# B&R Automation Studio project MotionTestBenchMaster
Automation Studio 4.2.12.129 SP

## Logical view

Binary libraries used (declarations not repeated): ArEventLog, AsARCfg, AsArProf, AsArSdm, AsEthIP, AsIecCon, AsICMP, AsIODiag, AsMath, asstring, AsTCP, astime, AsUDP, brsystem, DataObj, FileIO, LoopConR 4.01.0, operator, powerlnk, runtime, standard, sys_lib, AsMem, AsBrStr, dvframe, MpRecipe 1.61.0, AsEPL, MpCom 1.61.0, AsXml, AsIOLink, AsIOAcc, Acp10man 3.17.2, Acp10par 3.17.2, NcGlobal 3.17.2, Acp10sim 3.17.2, Acp10_MC 3.17.2, MpAxis 1.61.0, MpAlarmX 1.61.0, MpWebXs 1.61.0

### Package Logical/00_AID - Aid memory: memorie ausiliarie al programma

### Program Logical/00_AID/AID (IEC) - AID Main Program - C#3 - 1.6ms

#### AID.st - Cyclic code
```iecst
PROGRAM _INIT
	AID.DataOut.ProjectType	:= CST_AID_ProjectMachine;
END_PROGRAM

PROGRAM _CYCLIC
	TimeAndBlink;

	Beacon_SidelStandard;

	PbLight;

	AID.DataOut.Reset		:= IO_PB_ResetOp.ON;//v4 200.2.0
	IO_SkdReset.DO_Output	:= AID.DataOut.Reset;

	IF EDGEPOS(IO_PB_ResetOp.ON) THEN
		AID.DataOut.OperatorPresence	:= TRUE;
	END_IF
END_PROGRAM
```

#### Variables.var - Local variables
```iecst
VAR
	TMR_TP_HornAlarmStop : TP_Reset;
	VAR_AlarmLightReset : BOOL;
	VAR_CriticalLight : BOOL;
	VAR_AlarmLight : BOOL;
	VAR_AlarmHorn : BOOL;
	FB_Blink_05Hz : FB_Blinker;
	FB_Blink_1Hz : FB_Blinker;
	FB_Blink_4Hz : FB_Blinker;
	FB_Blink_2Hz : FB_Blinker;
	VAR_RedLightFix : BOOL;
	VAR_RedLightFlash : BOOL;
	VAR_BlueLightFix : BOOL;
	VAR_BlueLightFlash : BOOL;
	TMR_TON_InterCpuCycleOk : TON;
END_VAR
```

### Global.typ - Global data types
```iecst
(*HMI/IO BOTTON TYPE*)

TYPE
	PB_Type : 	STRUCT  (*Push button (ON-OFF;) 0=OFF - 1=ON*)
		Enable : BOOL; (*State: Command Enabled*)
		LampON : BOOL; (*State: Lamp Command ON*)
		Blink : BOOL; (*State: Blink LampOn*)
		Visibility : BOOL; (*Configuration: Present*)
		ON : BOOL; (*Command: Push Button ON*)
	END_STRUCT;
	SS2P_Type : 	STRUCT  (*Selector 2 position (Auto-Man; ON-OFF;) 0=Auto/OFF - 1=Man/ON*)
		Enable : BOOL; (*State: Command Enabled*)
		LampON : BOOL; (*State: Lamp Command ON*)
		Blink : BOOL; (*State: Blink LampOn*)
		Visibility : BOOL; (*Configuration: Present*)
		ON : BOOL; (*Command: Selector Button ON*)
	END_STRUCT;
	SS3P_Type : 	STRUCT  (*Selector 3 position (Auto-0-Man)*)
		Enable : BOOL; (*State: Command Enabled*)
		LampON : BOOL; (*State: Lamp Command ON*)
		Blink : BOOL; (*State: Blink LampOn*)
		Visibility : BOOL; (*Configuration: Present*)
		Auto : BOOL := TRUE; (*Command: Automatic Mode*)
		Man : BOOL; (*Command: Manual Mode ON*)
	END_STRUCT;
	CmdBarPB_Type : 	STRUCT  (*Push button (ON-OFF;) 0=OFF - 1=ON*)
		Enable : BOOL; (*State: Command Enabled*)
		LampON : BOOL; (*State: Lamp Command ON*)
		Blink : BOOL; (*State: Blink LampOn*)
		Visibility : BOOL; (*Configuration: Present*)
		ON : BOOL; (*Command: Push Button ON*)
		Command : BOOL; (*Command: Push Button On from HMI OR Command from ITC*)
	END_STRUCT;
	SS2PCustom_Type : 	STRUCT  (*V4.A.A.1.6.13*)
		Enable : BOOL; (*State: Command Enabled*)
		LampON : BOOL; (*State: Lamp Command ON*)
		Blink : BOOL; (*State: Blink LampOn*)
		Visibility : BOOL; (*Configuration: Present*)
		ON : BOOL; (*Command: Selector Button ON*)
		Description : STRING[25];
	END_STRUCT;
END_TYPE

(*OUTPUT TYPE*)

TYPE
	IO_Beacon_Type : 	STRUCT
		DO_LightGreen : BOOL;
		DO_LightYellow : BOOL;
		DO_LightBlue : BOOL;
		DO_LightWhite : BOOL;
		DO_LightRed : BOOL;
		DO_Horn : BOOL;
	END_STRUCT;
END_TYPE
```

### Alarm.var - Alarms structure declaration
```iecst
VAR
	ALR : ARRAY[1..8000] OF AlarmCmd_Type;
	ALR_OldStatus : ARRAY[1..8000] OF BOOL;
	ALR_CFG : ARRAY[1..8000] OF AlarmCFG_Type;
	VAR_ALR_FirstAlertAlarmActive : AlarmCFG_Type; (*V4.A.A.1.7.0*)
	VAR_ALR_FirstCriticalAlarmActive : AlarmCFG_Type; (*V4.A.A.1.7.0*)
	VAR_ALR_FirstAlarmActive : AlarmCFG_Type; (*V4.A.A.1.7.0*)
	VAR_ALR_FirstExternalAlarmActive : AlarmCFG_Type; (*V4.A.A.1.7.0*)
	VAR_ALR_FirstExtCritAlarmActive : AlarmCFG_Type; (*V4.A.A.1.7.0*)
	VAR_ALR_FirstExtAlertAlarmActive : AlarmCFG_Type; (*V4.A.A.1.7.0*)
	VAR_ALR_FirstCsAlarmActive : AlarmCFG_Type; (*V4.A.A.1.7.0*)
	VAR_ALR_FirstCsExtAlarmActive : AlarmCFG_Type; (*V4.A.A.1.7.5a*)
	VAR_ALR_CriticalAcknoledgeReq : BOOL;
	VAR_ALR_AlarmAcknoledgeReq : BOOL;
	VAR_AlarmActionOper : ActionSum_Type; (*V4.A.A.1.6.13*)
	VAR_FMC_AlarmActionOper : ActionSum_Type;
	VAR_SKD_AlarmActionOper : ActionSum_Type;
END_VAR
```

### Package Logical/00_AID/IO - Input/Output declaration

### IO_AID.var
```iecst
VAR
	IO_SkdReset : IO_Digital_OUT_Type;
	IO_InterCpu_NettimeSoC : DINT;
	IO_InterCpu_CicleOk : BOOL;
END_VAR
```

### IO_CAP.var
```iecst
(*MOTORS*)
VAR
	IO_206MMR : IO_Motor_Type; (*Head rotation motor*)
	IO_206MMRBrake : IO_Motor_Type; (*Head rotation motor brake*)
	IO_207MMR : IO_Motor_Type; (*Hopper motor chute 1*)
	IO_211MMR : IO_Motor_Type; (*Buffer rotation motor2 v1.7.4*)
	IO_212MMR : IO_Motor_Type; (*Buffer rotation motor*)
	IO_213MMR : IO_Motor_Type; (*Head rotation motor fun*)
	IO_214MMR : IO_Motor_Type; (*Hopper motor chute 2*)
	IO_215MMR : IO_Motor_Type; (*Hopper motor chute 3*)
	IO_229MMR : IO_Motor_Type; (*Adjustment panel motor //V4.A.A.1.6.11*)
	IO_229MMR_Start : IO_SiriusStarter_Type; (*Adjustment panel motor //V4.A.A.1.6.11*)
	IO_230MMR : IO_Motor_Type; (*Dust removal motor on caps channel*)
	IO_231MMR : IO_Motor_Type; (*Dust removal motor on buffer //V4.A.A.1.6.11*)
	IO_202GPE : IO_GreasingPump_Type; (*Capper Greasing Motor*)
	IO_203GPE : IO_GreasingPump_Type; (*Capper Greasing Motor2 //V4.A.A.1.6.11*)
END_VAR
(*IONIZER*)
VAR
	IO_201DRC : IO_Motor_Type; (*Hopper motor chute 2*)
	IO_201DRC_SwitchFeedback : IO_Digital_IN_Type;
END_VAR
(*UV LAMP*)
VAR
	IO_201LLC : IO_Motor_Type; (*UV lamp Chute 1*)
	IO_202LLC : IO_Motor_Type; (*UV lamp Chute 2*)
	IO_203LLC : IO_Motor_Type; (*UV lamp Chute 3*)
END_VAR
(*DRIVERS*)
VAR
	IO_VFD_206MMR : IO_PLK_Danfoss_Drive_Type; (*Head rotation motor*)
	IO_VFD_207MMR : IO_PLK_Danfoss_Drive_Type; (*Hopper motor chute 1*)
	IO_VFD_230MMR : IO_PLK_Danfoss_Drive_Type; (*Dust remover motor*)
	IO_VFD_231MMR : IO_PLK_Danfoss_Drive_Type; (*Dust remover motor2 v1.7.4*)
	IO_VFD_211MMR : IO_PLK_Danfoss_Drive_Type; (*Buffer rotation motor2 v1.7.4*)
	IO_VFD_213MMR : IO_PLK_Danfoss_Drive_Type; (*Head rotation motor fun*)
	IO_VFD_212MMR : IO_PLK_Danfoss_Drive_Type; (*Buffer rotation motor*)
	IO_VFD_214MMR : IO_PLK_Danfoss_Drive_Type; (*Hopper motor chute 2*)
	IO_VFD_215MMR : IO_PLK_Danfoss_Drive_Type; (*Hopper motor chute 3*)
END_VAR
(*VALVES*)
VAR
	IO_201CPC : IO_Valve_Type; (*EV chute 1 caps release*)
	IO_202CPC : IO_Valve_Type; (*EV chute 2 caps release*)
	IO_205CPC : IO_Valve_Type; (*EV caps block chute 1*)
	IO_206CPC : IO_Valve_Type; (*EV caps block chute 2*)
	IO_207CPC : IO_Valve_Type; (*EV cap discharge door*)
	IO_212CPC : IO_Valve_Type; (*EV open buffer discharge door*)
	IO_213CPC : IO_Valve_Type; (*EV buffer lifting*)
	IO_214CPC : IO_Valve_Type; (*EV buffer lock*)
	IO_215CPC : IO_Valve_Type; (*EV lock size change guide*)
	IO_216CPC : IO_Valve_Type; (*EV 3 size change guide*)
	IO_217CPC : IO_Valve_Type; (*EV 4 size change guide*)
	IO_218CPC : IO_Valve_Type; (*EV sport size change guide*)
	IO_219CPC : IO_Valve_Type; (*EV open channel discharge door*)
	IO_220CPC : IO_Valve_Type; (*FREE v1.7.6*)
	IO_221CPC : IO_Valve_Type; (*EV chute 3 caps release*)
	IO_222CPC : IO_Valve_Type; (*EV caps block chute 3*)
	IO_223CPC : IO_Valve_Type; (*EV buffer vibrator*)
	IO_224CPC : IO_Valve_Type; (*EV cam position*)
	IO_225CPC : IO_Valve_Type; (*EV cam locking*)
	IO_226CPC : IO_Valve_Type; (*EV opening door UV Lamp A  V. 1.1*)
	IO_227CPC : IO_Valve_Type; (*EV  Block Caps Outlet Chute 1*)
	IO_228CPC : IO_Valve_Type; (*EV transfer Starwheel air soleniod valve DA VERIFICARE*)
	IO_229CPC : IO_Valve_Type; (*EV transfer Starwheel air soleniod valve DA VERIFICARE*)
	IO_232CPC : IO_Valve_Type; (*EV opening door UV Lamp B  V. 1.1*)
	IO_233CPC : IO_Valve_Type; (*EV opening door UV Lamp B  //V4.A.A.1.6.12*)
	IO_234CPC : IO_Valve_Type; (*EV Caps Ejection Cap Feeder   V4.A.A.1.7.1*)
	IO_235CPC : IO_Valve_Type; (*EV Caps Block Outlet Chuter2 //v1.7.4*)
	IO_236CPC : IO_Valve_Type; (*v1.7.4*)
	IO_237CPC : IO_Valve_Type; (*v1.7.4*)
	IO_238CPC : IO_Valve_Type; (*v1.7.4*)
	IO_201EVC : IO_Valve_Type; (*Air blowing for cap release 1 V 1.6*)
	IO_203EVC : IO_Valve_Type; (*Air blowing for cap release 2 V 1.6*)
	IO_207EVC : IO_Valve_Type; (*Air blowing for cap release 3 V 1.6*)
	IO_209EVC : IO_Valve_Type; (*FREE V1.6*)
	IO_210EVC : IO_Valve_Type; (*Air blowing for buffer emptying*)
	IO_211EVC : IO_Valve_Type; (*Buffer air blowing for caps release*)
	IO_212EVC : IO_Valve_Type; (*Air blowing for chute emptying*)
	IO_213EVC : IO_Valve_Type; (*Air blowing caps ionizer chute 1*)
	IO_214EVC : IO_Valve_Type; (*Air blowing caps ionizer chute 2*)
	IO_215EVC : IO_Valve_Type; (*Air blowing caps ionizer chute 3*)
	IO_216EVC : IO_Valve_Type; (*Air blowing for chute emptying by PeP*)
	IO_227EVC : IO_Valve_Type; (*v1.7.4*)
	IO_228EVC : IO_Valve_Type; (*v1.7.4*)
	IO_229EVC : IO_Valve_Type; (*v1.7.4*)
	IO_203EVF : IO_Valve_Type; (*Air blowing caps (Drying)*) (*IO_AVC : ARRAY[MIN_CFG_AVC..MAX_CFG_AVC] OF IO_Valve_Type; Caps Treatment Valves v4.A.A.1.7.0*)
END_VAR
(*SENSOR*)
VAR
	IO_201DSC : IO_Digital_IN_Type; (*Caps/crowns release check*)
	IO_202DSC : IO_Digital_IN_Type; (*Low level caps/crowns presence chute 1*)
	IO_204DSC : IO_Digital_IN_Type; (*Head 1 sensor*)
	IO_205DSC : IO_Digital_IN_Type; (*Lack of caps (Quibuf infeed)*)
	IO_210DSC : IO_Digital_IN_Type; (*Cap Overturned hight Cap Feeder  V4.A.A.1.7.1*)
	IO_211DSC : IO_Digital_IN_Type; (*Cap Overturned low Cap Feeder  V4.A.A.1.7.1*)
	IO_216DSC : IO_Digital_IN_Type; (*Low level caps/crowns presence chute 2*)
	IO_217DSC : IO_Digital_IN_Type; (*Low level caps/crowns presence chute 3*)
	IO_218DSC : IO_Digital_IN_Type; (*Upside down caps check chute 1 high*)
	IO_219DSC : IO_Digital_IN_Type; (*Upside down caps check chute 1 low*)
	IO_220DSC : IO_Digital_IN_Type; (*Upside down caps check chute 2 high*)
	IO_221DSC : IO_Digital_IN_Type; (*Upside down caps check chute 2 low*)
	IO_222DSC : IO_Digital_IN_Type; (*Upside down caps check chute 3 high*)
	IO_223DSC : IO_Digital_IN_Type; (*Upside down caps check chute 3 low*)
	IO_224DSC : IO_Digital_IN_Type; (*Ionizer pressure switch chute 1*)
	IO_225DSC : IO_Digital_IN_Type; (*Ionizer pressure switch chute 2*)
	IO_226DSC : IO_Digital_IN_Type; (*Ionizer pressure switch chute 3*)
	IO_227DSC : IO_Digital_IN_Type; (*Lubrication door sensor*)
	IO_228DSC : IO_Digital_IN_Type; (*Fixed part lubrication check*)
	IO_229DSC : IO_Digital_IN_Type; (*Rotating part lubrication check*)
	IO_230DSC : IO_Digital_IN_Type; (*Lubrication pipe inserted sensor*)
	IO_231DSC : IO_Digital_IN_Type; (*Turret cam position analog sensor*)
	IO_232DSC : IO_Digital_IN_Type; (*Caps buffer full*)
	IO_233DSC : IO_Digital_IN_Type; (*Caps channel discharge gate sensor*)
	IO_234DSC : IO_Digital_IN_Type; (*Lubrication phase sensor*)
	IO_235DSC : IO_Digital_IN_Type; (*Buffer in high position*)
	IO_236DSC : IO_Digital_IN_Type; (*Buffer in low position*)
	IO_237DSC : IO_Digital_IN_Type; (*Buffer lock inserted*)
	IO_238DSC : IO_Digital_IN_Type; (*Caps buffer max level chute 1*)
	IO_239DSC : IO_Digital_IN_Type; (*Caps buffer max level chute 2*)
	IO_240DSC : IO_Digital_IN_Type; (*Caps buffer max level chute 3*)
	IO_241DSC : IO_Digital_IN_Type; (*Hopper level chute 1*)
	IO_242DSC : IO_Digital_IN_Type; (*Hopper level chute 2*)
	IO_243DSC : IO_Digital_IN_Type; (*Hopper level chute 3*)
	IO_244DSC : IO_Digital_IN_Type; (*Max level caps/crowns chute 1*)
	IO_245DSC : IO_Digital_IN_Type; (*Max level caps/crowns chute 2*)
	IO_246DSC : IO_Digital_IN_Type; (*Max level caps/crowns chute 3*)
	IO_247DSC : IO_Digital_IN_Type; (*Medium level caps/crowns chute 1*)
	IO_248DSC : IO_Digital_IN_Type; (*Medium level caps/crowns chute 2*)
	IO_249DSC : IO_Digital_IN_Type; (*Medium level caps/crowns chute 3*)
	IO_250DSC : IO_Digital_IN_Type; (*Side door hopper sport*)
	IO_251DSC : IO_Digital_IN_Type; (*Top door hopper sport*)
	IO_252DSC : IO_Digital_IN_Type; (*Uv lamp door*)
	IO_253DSC : IO_Digital_IN_Type; (*Sensore carter posteriore*)
	IO_254DSC : IO_Digital_IN_Type; (*Sensore di fase per lubrificazione*)
	IO_255DSC : IO_Digital_IN_Type; (*Sensore di lubrificazione della parte fissa*)
	IO_256DSC : IO_Digital_IN_Type; (*Sensore di lubrificazione della parte rotante*)
	IO_257DSC : IO_Digital_IN_Type; (*Sensore di inserimento del raccordo di lubrificazione della parte rotante *)
	IO_258DSC : IO_Digital_IN_Type; (*Sensore carter superiore  //V4.A.A.1.6.11*)
	IO_259DSC : IO_Digital_IN_Type; (*Sensore di lubrificazione rotazione teste //V4.A.A.1.6.11*)
	IO_260DSC : IO_Digital_IN_Type; (*Sensore di inserimento del raccordo di lubrificazione della parte rotante riduttore rotazione teste //V4.A.A.1.6.11*)
	IO_261DSC : IO_Digital_IN_Type; (*Sensore limite minimo posizione pannello //V4.A.A.1.6.11*)
	IO_262DSC : IO_Digital_IN_Type; (*Sensore zero encoder //V4.A.A.1.6.11*)
	IO_263DSC : IO_Digital_IN_Type; (*Sensore limite massimo posizione pannello //V4.A.A.1.6.11*)
	IO_264DSC : IO_Digital_IN_Type; (*Caps/Crown release check on bottle   //V4.A.A.1.6.12h*)
	IO_266DSC : IO_Digital_IN_Type; (*Flow Cap Control //v1.7.4*)
	IO_267DSC : IO_Digital_IN_Type; (*v1.7.5*)
	IO_268DSC : IO_Digital_IN_Type; (*v1.7.5*)
	IO_270DSC : IO_Digital_IN_Type; (*Caps Belt Sensor  //v1.7.4*)
	IO_ST3B : IO_Analog_IN_Type; (*Sensore temperatura motore//V4.A.A.1.6.12*)
	IO_ST3A : IO_Analog_IN_Type; (*Sensore temperatura motore//V4.A.A.1.6.12*)
END_VAR
(*COUNTERS*)
VAR
	IO_201DGC : IO_IncrementalEncoder; (*Incremental Encoder adjustment panel //V4.A.A.1.6.11*)
END_VAR
(*PB*)
VAR
	IO_PB_BufferUp : PB_Type;
	IO_PB_BufferDown : PB_Type;
END_VAR
(*MOTORS EQUATORQUE & HRM*)
VAR
	IO_BrushHead : IO_Motor_Type; (*Outfeed Conveyor Motor V4.A.A.1.6.12*)
END_VAR
(*DIGITAL OUTPUT*)
VAR
	IO_CAP_24Vdc_OK : IO_Digital_OUT_Type; (*v1.5*)
	IO_BottlePresence : IO_Digital_OUT_Type; (*v1.5*)
	IO_CapsRequest : IO_Digital_OUT_Type; (*v1.7.4 Richiesta capsule all'elevatore*)
END_VAR
```

### IO_CRW.var
```iecst
(*VALVES*)
VAR
	IO_230CPC : IO_Valve_Type; (*EV chute 1 crowns release*)
	IO_231CPC : IO_Valve_Type; (*EV chute 2 crowns release*)
	IO_231EVC : IO_Valve_Type;
	IO_205EVC : IO_Valve_Type; (*EXTRACTOR BLOWER CLEANING*)
	IO_274DSC : IO_Digital_IN_Type; (*Master nuovo*)
END_VAR
```

### IO_CSR.var
```iecst
(*Master nuovo*)
VAR
	IO_204CPC : IO_Valve_Type; (*EV crowner lift block*)
	IO_LTK : ARRAY[MIN_CFG_LTx..MAX_CFG_LTx] OF IO_Analog_IN_Type;
	IO_3281M1 : IO_Motor_FwBw_Type;
	IO_3281M1_Cmd : IO_Digital_OUT_Type;
	IO_2806M1 : IO_Motor_FwBw_Type;
	IO_2806M1_Cmd : IO_Digital_OUT_Type;
	IO_2808M1 : IO_Motor_FwBw_Type;
	IO_2806M1_Brake : IO_Motor_Type;
	IO_2809M2_Brake : IO_Motor_Type;
	IO_2809M2 : IO_Motor_FwBw_Type;
	IO_RnsLiftFC280 : IO_MotorFC280_Type; (*Rinser Lift*)
	IO_VFD_RnsLiftFC280 : IO_PLK_DanfossFC280_Drive_Type; (*Rinser Lift VFD*)
	IO_TnkLiftFC280 : IO_MotorFC280_Type;
	IO_VFD_TnkLiftFC280 : IO_PLK_DanfossFC280_Drive_Type; (*Outfeed Conveyor VFD*)
	IO_2768U0 : IO_Motor_FwBw_Type;
	IO_2768U0_Store : IO_Digital_OUT_Type;
	IO_202CPB : IO_Valve_Type; (*Containers sectors block (X: Block / Y: Unblock)*)
	IO_212DSB : IO_Digital_IN_Type; (*Third element perso part sensor*)
	IO_213DSB : IO_Digital_IN_Type; (*Third element perso part sensor - Ferrum Guide Presence in Carousel Outlet*)
	IO_CSR_SCU : IO_CSR_SCU_Type;
	IO_CSR_FlrShaftSensorCtrl1 : IO_Digital_IN_Type;
	IO_CSR_FlrShaftSensorCtrl2 : IO_Digital_IN_Type;
	IO_CSR_RnsShaftSensorCtrl1 : IO_Digital_IN_Type;
	IO_CSR_RnsShaftSensorCtrl2 : IO_Digital_IN_Type;
	IO_YV26 : IO_Valve_Type;
	IO_YV39 : IO_Valve_Type;
	IO_SQ26 : IO_Digital_IN_Type;
	IO_SQ45A2 : IO_Digital_IN_Type;
	IO_SQ45A1 : IO_Digital_IN_Type;
	IO_SQ70 : IO_Digital_IN_Type;
	IO_SQ5 : IO_Digital_IN_Type;
	IO_SQ40 : IO_Digital_IN_Type;
	IO_SQ6 : IO_Digital_IN_Type;
	IO_3565S5 : IO_Digital_IN_Type;
	IO_3565S7 : IO_Digital_IN_Type;
	IO_CapChannelPresent : IO_Digital_IN_Type;
END_VAR
(*SIKO*)
VAR
	IO_SIKO_AX2_SafetyEnable : IO_Digital_IN_Type := (DI_Input:=TRUE);
	IO_SIKO_AX1_SafetyEnable : IO_Digital_IN_Type := (DI_Input:=TRUE);
	IO_SIKO_AX1_Overload : IO_Digital_IN_Type := (DI_Input:=TRUE);
	IO_SIKO_AX2_Overload : IO_Digital_IN_Type := (DI_Input:=TRUE);
	IO_SIKO_AX1_ModuleOK : IO_Digital_IN_Type; (*Module Ok: Put this IO in The IoMap*)
	IO_SIKO_AX2_ModuleOK : IO_Digital_IN_Type; (*Module Ok: Put this IO in The IoMap*)
	IO_SIKO_AX1 : SIKO_COM_Type;
	IO_SIKO_AX2 : SIKO_COM_Type;
	IO_238DSE : IO_Digital_IN_Type; (*Outlet Conveyor Height Sensor*)
	IO_243DSE : IO_Digital_IN_Type; (*Outlet Conveyor Body Guide Presence*)
END_VAR
```

### IO_DMC.var
```iecst
VAR
	IO_210EVF : IO_Valve_Type; (*master nuovo*)
	IO_211EVF : IO_Valve_Type; (*master nuovo*)
	IO_RollSafety1 : IO_Dmc_Type;
	IO_RollSafety2 : IO_Dmc_Type;
	IO_DmcDevice : IO_Dmc_Type;
	IO_205DSF : IO_Digital_IN_Type; (*Dummy container inserted*)
END_VAR
```

### IO_FMC.var
```iecst
VAR
	IO_PB_FmcStartFilling : PB_Type; (*Manual filling start from Hw button*)
	IO_PB_FmcStopFilling : PB_Type; (*Manual filling stop from Hw button*)
	IO_PB_FmcStep : PB_Type; (*Single step from Hw button*)
END_VAR
```

### IO_GNS.var
```iecst
(*VALVES*)
VAR
	IO_201EVR : IO_Valve_Type; (*Ev MB05 Cooling*)
	IO_204EVF : IO_Valve_Type; (*Ev Pilot valve air (X: Discharge / Y: Charge)*)
	IO_205EVF : IO_Valve_Type;
END_VAR
(*SENSORS*)
VAR
	IO_204PSF : IO_Digital_IN_Type; (*Carousel air pressure switch*)
	IO_201PTF : IO_Analog_IN_Type; (*Carousel air pressure sensor*)
	IO_205PTF : IO_Analog_IN_Type; (*Carousel air pressure sensor*)
	IO_206PTF : IO_Analog_IN_Type; (*Carousel air pressure sensor*)
	IO_204PTF : IO_Analog_IN_Type; (*Carousel air pressure sensor*)
	IO_235DSE : IO_Digital_IN_Type; (*Cop mode Conveyor Outlet*)
	IO_239DSE : IO_Digital_IN_Type; (*Production mode Transfer Inlet*)
	IO_240DSE : IO_Digital_IN_Type; (*Cop mode Transfer Inlet*)
	IO_242DSE : IO_Digital_IN_Type; (*Production mode Conveyor Outlet*)
	IO_ContainerBurst1 : IO_Digital_IN_Type; (*ContainerBurst#1*)
	IO_ContainerBurst2 : IO_Digital_IN_Type; (*ContainerBurst#2 *)
	IO_201QTB : IO_Analog_IN_Type; (*Basement Air Control - CO2 Sensor //v1.7.4*)
	IO_201QTB_Warning : IO_Digital_IN_Type; (*Basement Air Control - CO2 Sensor Warning //v1.7.4*)
	IO_201QTB_Alarm : IO_Digital_IN_Type; (*Basement Air Control - CO2 Sensor Alarm//v1.7.4*)
	IO_201QTE : IO_Analog_IN_Type; (*Filler Air Control - CO2 Sensor //v1.7.4*)
	IO_201QTE_Warning : IO_Digital_IN_Type; (*FIller Air Control - CO2 Sensor Warning //v1.7.4*)
	IO_201QTE_Alarm : IO_Digital_IN_Type; (*Filler Air Control - CO2 Sensor Alarm//v1.7.4*)
	IO_202QTB : IO_Analog_IN_Type; (*Basement Air Control - Ozozne Sensor //v1.7.4*)
	IO_202QTB_Warning : IO_Digital_IN_Type; (*Basement Air Control - Ozozne Sensor Warning //v1.7.4*)
	IO_202QTB_Alarm : IO_Digital_IN_Type; (*Basement Air Control - Ozozne Sensor Alarm//v1.7.4*)
	IO_202QTE : IO_Analog_IN_Type; (*Filler Air Control - Ozozne Sensor //v1.7.4*)
	IO_202QTE_Warning : IO_Digital_IN_Type; (*Filler Air Control - Ozozne Sensor Warning //v1.7.4*)
	IO_202QTE_Alarm : IO_Digital_IN_Type; (*Filler Air Control - Ozozne Sensor Alarm//v1.7.4*)
END_VAR
(*INSTRUMENTS - DIGITAL*)
VAR
	IO_MB05_Cooling : IO_Cooling_Type; (*MB05 Cooling*)
	IO_MB05_Overload : IO_Digital_IN_Type := (DI_Input:=TRUE); (*MB05 Auxiliary circuit ON*)
	IO_MB15_Cooling : IO_Cooling_Type; (*MB15 Cooling v1.62*)
	IO_MB15_Overload : IO_Digital_IN_Type := (DI_Input:=TRUE); (*MB15 Auxiliary circuit ON*)
	IO_MB25_Overload : IO_Digital_IN_Type := (DI_Input:=TRUE); (*MB25 Auxiliary circuit ON*)
	IO_MC01_Cooling : IO_Cooling_Type; (*MC01 Cooling*)
	IO_MC01_Overload : IO_Digital_IN_Type := (DI_Input:=TRUE); (*MC01 Auxiliary circuit ON*)
	IO_MC02_Cooling : IO_Cooling_Type; (*MC02 Cooling*)
	IO_MC02_5VOverload : IO_Digital_IN_Type := (DI_Input:=TRUE); (*MC02 Auxiliary circuit ON*)
	IO_MC02_Overload : IO_Digital_IN_Type := (DI_Input:=TRUE); (*MC02 Auxiliary circuit ON*)
	IO_MC04_Cooling : IO_Cooling_Type; (*MC04 Cooling*)
	IO_MC04_Overload : IO_Digital_IN_Type := (DI_Input:=TRUE); (*MC04 Auxiliary circuit ON*)
	IO_MC04_CabinetDoorsUnlockFbk : IO_Digital_IN_Type; (*MC04 Cabinet Doors Unlock Feedback*)
	IO_MC04_CabinetDoorsUnlockReq : IO_Digital_IN_Type; (*MC04 Cabinet Doors Unlock Request*)
	IO_MC04_DoorCabinetOpened : IO_Digital_IN_Type := (DI_Input:=TRUE); (*MC04 Cabinet Door Opened*)
	IO_MC07_Cooling : IO_Cooling_Type; (*MC07 Cooling*)
	IO_MC07_Overload : IO_Digital_IN_Type := (DI_Input:=TRUE); (*MC07 Auxiliary circuit ON*)
	IO_MC07_DoorCabinetOpened : IO_Digital_IN_Type := (DI_Input:=TRUE); (*MC07 Cabinet Door Opened*)
	IO_MC19_Overload : IO_Digital_IN_Type := (DI_Input:=TRUE); (*MC19 Auxiliary circuit ON*)
	IO_MC19_DoorCabinetOpened : IO_Digital_IN_Type := (DI_Input:=TRUE); (*MC19 Cabinet Door Opened*)
	IO_MC29_Cooling : IO_Cooling_Type; (*MC29 Cooling  //v999hema*)
	IO_MC29_Overload : IO_Digital_IN_Type := (DI_Input:=TRUE); (*MC29 Auxiliary circuit ON //v999hema*)
	IO_MC29_DoorCabinetOpened : IO_Digital_IN_Type := (DI_Input:=TRUE); (*MC29 Cabinet Door Opened VRMA*)
	IO_CapFeederOverload : IO_Digital_IN_Type := (DI_Input:=TRUE); (*CapFeeder Overload ON*)
	IO_OptifeedOverload : IO_Digital_IN_Type := (DI_Input:=TRUE); (*Optifeed Overload ON //V4.A.A.1.6.11*)
	IO_UPS : IO_UPS_Type;
END_VAR
(*OUTPUT*)
VAR
	IO_FlrBeacon : IO_Beacon_Type;
END_VAR
```

### IO_ITC.var
```iecst
VAR
	IO_PB_LbStart : PB_Type; (*Labeller start Hw button*)
	IO_PB_LbStop : PB_Type; (*Labeller stop Hw button*)
END_VAR
(*HARDWARE\DP COMMUNICATION*)
VAR
	IO_ITC : IO_ITC_Type;
END_VAR
```

### IO_MAU.var
```iecst
(*MOTORS*)
VAR
	IO_201GPE : IO_GreasingPump_Type; (*MACHINE GREASING PUMP*)
END_VAR
(*OUTPUT*)
VAR
	IO_MachineLight : IO_Digital_OUT_Type;
END_VAR
(*PRESSURIZER*)
VAR
	IO_FanBase : IO_FanMain_Type;
	IO_FanFiller : IO_FanMain_Type;
	IO_FanRinser : IO_FanMain_Type;
	IO_FanTransfer : IO_FanMain_Type;
END_VAR
(*PLC*)
VAR
	IO_CPU : IO_CPU_Type;
END_VAR
(*LIFT CONTAINERS*)
VAR
	IO_203PSF : IO_Digital_IN_Type;
	IO_205RVF : IO_Analog_IN_OUT_Type;
	IO_203RVF : IO_Analog_IN_OUT_Type;
	IO_206DSF : IO_Digital_IN_Type; (*Filling valve 1 sensor*)
	IO_FSF : ARRAY[MIN_CFG_FSx..MAX_CFG_FSx] OF IO_Digital_IN_Type;
END_VAR
```

### IO_MNM.var
```iecst
VAR
	IO_PB_FlStart : PB_Type; (*Filler start Hw button*)
	IO_PB_FlStop : PB_Type := (ON:=TRUE); (*Filler stop Hw button*)
	IO_PB_ResetOp : PB_Type; (*Reset Hw button*)
	IO_PB_ResetFwIn : PB_Type; (*Reset Hw button*)
	IO_PB_ResetFwOut : PB_Type; (*Reset Hw button*)
	IO_PB_ResetBkIn : PB_Type; (*Reset Hw button*)
	IO_PB_ResetBkOut : PB_Type; (*Reset Hw button*)
	IO_KochModuleOk : IO_Digital_IN_Type;
END_VAR
(*MOTORS*)
VAR
	IO_InCvrFC280 : IO_MotorFC280_Type; (*Outfeed Conveyor Motor*) (*Master nuovo*)
	IO_OutCvrFC280 : IO_MotorFC280_Type; (*Outfeed Conveyor Motor*) (*Master nuovo*)
	IO_InCvr : IO_Motor_Type; (*Outfeed Conveyor Motor*) (*Master nuovo*)
	IO_OutCvr : IO_Motor_Type; (*Outfeed Conveyor Motor*)
END_VAR
(*DRIVERS*)
VAR
	IO_VFD_InCvrFC280 : IO_PLK_DanfossFC280_Drive_Type; (*Outfeed Conveyor VFD*) (*Master nuovo*)
	IO_VFD_OutCvrFC280 : IO_PLK_DanfossFC280_Drive_Type; (*Outfeed Conveyor VFD*) (*Master nuovo*)
	IO_VFD_InCvr : IO_PLK_Danfoss_Drive_Type; (*Outfeed Conveyor VFD*) (*Master nuovo*)
	IO_VFD_OutCvr : IO_PLK_Danfoss_Drive_Type; (*Outfeed Conveyor VFD*)
END_VAR
(*DIGITAL INSTUMENTS*)
VAR
	IO_241DSE : IO_Digital_IN_Type; (*Caps Discharge*)
	IO_230DSE : IO_Digital_IN_Type; (*Spot safety*)
	IO_236DSE : IO_Digital_IN_Type; (*Outlet obstructed*)
	IO_217DSR : IO_Digital_IN_Type; (*Machine upper part access tool position control V4.A.A.1.6.13*)
	IO_296CPB_I : IO_Digital_IN_Type; (*V4.A.A.1.7.0 RInser Bypass Control*)
	IO_297CPB_I : IO_Digital_IN_Type; (*V4.A.A.1.7.0 Rinser Bypass Control*)
	IO_224DSB : IO_Digital_IN_Type; (*Doser Bypass Control RMH017*)
	IO_225DSB : IO_Digital_IN_Type; (*Doser Bypass Control *)
	IO_226DSB : IO_Digital_IN_Type; (*Doser Bypass Control *)
	IO_227DSB : IO_Digital_IN_Type; (*Doser Bypass Control *)
END_VAR
(*MOTION Feedback*)
VAR
	IO_MNM_MotionFan : IO_MotionFanMachine_Type;
	IO_MNM_PowerSupply1Overload : IO_Digital_IN_Type := (DI_Input:=TRUE);
	IO_MNM_PowerSupply2Overload : IO_Digital_IN_Type := (DI_Input:=TRUE);
END_VAR
(*INLET CANS SENSOR*)
VAR
	IO_InletSafetyLow1 : IO_Digital_IN_Type;
	IO_InletSafetyHigh1 : IO_Digital_IN_Type;
	IO_InletSafetyLow2 : IO_Digital_IN_Type;
	IO_InletSafetyHigh2 : IO_Digital_IN_Type;
END_VAR
(*INLET CONTAINER RESET*)
(*Master nuovo*)
VAR
	IO_PB_ResetInlet1 : PB_Type; (*Master nuovo*)
	IO_PB_ResetInlet2 : PB_Type; (*Master nuovo*)
END_VAR
(* *)
VAR
	IO_LimitTorqueBlowerTransfer : IO_Digital_IN_Type := (DI_Input:=TRUE);
END_VAR
```

### IO_MC.var
```iecst
VAR
	IO_MCRaw : IO_MCRaw_Type;
	ITC_Motion_ExtEncModuleOk : BOOL;
	ITC_Motion_ExtEnc : DINT;
END_VAR
```

### IO_OPS.var
```iecst
VAR
	PO : PO_Safety_Type;
	PI : PI_Safety_Type;
	IO_OPS_Door : ARRAY[MIN_CFG_SafetyZone..MAX_CFG_SafetyZone,MIN_CFG_SafetyDoor..MAX_CFG_SafetyDoor] OF IO_OPS_Door_Type; (*1: Forward
2: Backward 1
3: Backward 2
4: Inlet Transfer Forward
5: Inlet Transfer Backward
6: Outlet Transfer Forward
7: Outlet Transfer Backward
8: Maintenance 1
9: Maintenance 2
10: Inlet Transfer Gate
11: Outlet Transfer Gate
12: Capper*)
	IO_OPS_Zone : ARRAY[MIN_CFG_SafetyZone..MAX_CFG_SafetyZone] OF IO_OPS_Zone_Type; (*1: Forward
2: Backward 1
3: Backward 2
4: Inlet Transfer Forward
5: Inlet Transfer Backward
6: Outlet Transfer Forward
7: Outlet Transfer Backward
8: Maintenance 1
9: Maintenance 2
10: Inlet Transfer Gate
11: Outlet Transfer Gate
12: Capper*)
	IO_OPS_JOG : ARRAY[MIN_CFG_SafetyJog..MAX_CFG_SafetyJog] OF IO_OPS_JOG_Type;
	IO_207EVF : IO_Valve_Type; (*Soffio Paratia automatica COP V4.A.A.1.6.12*)
	IO_208CPF : IO_Valve_Type; (*Paratia automatica COP V4.A.A.1.6.12*)
	IO_208DSFX : IO_Digital_IN_Type; (*Paratia automatica COP Aperta V4.A.A.1.6.12*)
	IO_208DSFY : IO_Digital_IN_Type; (*Paratia automatica COP Chiusa V4.A.A.1.6.12*)
	IO_209DSFX : IO_Digital_IN_Type; (*Paratia automatica COP Aperta V4.A.A.1.6.12*)
	IO_209DSFY : IO_Digital_IN_Type; (*Paratia automatica COP Chiusa V4.A.A.1.6.12*)
	IO_209EVF : IO_Valve_Type;
	IO_SS3P_Modality : IO_SS3PModality_Type;
	SI_SafeLogicModuleOk : BOOL;
	IO_Euchner_Key : IO_Digital_IN_Type; (*V1.3*)
	IO_Euchner_Strobe : IO_Digital_IN_Type; (*V1.3*)
	IO_Euchner_CodeA : IO_Digital_IN_Type; (*V1.3*)
	IO_Euchner_CodeB : IO_Digital_IN_Type; (*V1.3*)
	IO_Euchner_CodeC : IO_Digital_IN_Type; (*V1.3*)
	IO_Euchner_CodeD : IO_Digital_IN_Type; (*V1.3*)
	IO_PB_FlrSlowRun1 : PB_Type; (*V1.3*)
	IO_PB_FlrSlowRun2 : PB_Type; (*V1.3*)
	IO_PB_FlrSlowRun3 : PB_Type; (*V1.3*)
END_VAR
```

### IO_SFT.var
```iecst
(*SENSORS*)
(*ANOLOG SENSORS*)
VAR
	IO_203DSF : IO_Digital_IN_Type; (*Container presence outlet filler*)
	IO_202DSF : IO_Digital_IN_Type; (*Filler inlet container presence*)
	IO_208FSE : IO_Digital_IN_Type; (*Washing Ramp3 Flow-switch*)
	IO_207FSE : IO_Digital_IN_Type; (*Washing Ramp2 Flow-switch*)
	IO_ProductionSensorCheck1 : IO_Digital_IN_Type; (*Production Sensor Check For DMC Automatic*) (*Master nuovo*)
	IO_ProductionSensorCheck2 : IO_Digital_IN_Type; (*Production Sensor Check For DMC Automatic*) (*Master nuovo*)
	IO_ProductionSensorCheck3 : IO_Digital_IN_Type; (*Production Sensor Check For DMC Automatic*) (*Master nuovo*)
END_VAR
(*FLOW-SWITCHES*)
VAR
	IO_206FSE : IO_Digital_IN_Type; (*Washing Ramp1 Flow-switch*)
	IO_202EVR : IO_Valve_Type; (*Ev guide heater (VBS)*)
	IO_208CPB : IO_Valve_Type; (*Nob Nos 2° Treatment*)
	IO_207CPB : IO_Valve_Type; (*Nob Nos 1° Treatment*)
	IO_207CPF : IO_Valve_Type; (*Roller Security Cam*)
END_VAR
(*VALVES*)
VAR
	IO_201CPB : IO_Valve_Type; (*Inlet Bottle Block Bottle Stop*)
	IO_BurstCheck : ARRAY[0..2] OF IO_Digital_IN_Type; (*Container Burst Check 1*) (*Master nuovo*)
	IO_205DSB : IO_Digital_IN_Type; (*Doser outlet container presence*)
	IO_208DSF : IO_Digital_IN_Type; (*Rinser outlet container presence*)
	IO_DummyClock : IO_Digital_IN_Type; (*Rinser inlet container presence*)
	IO_207DSF : IO_Digital_IN_Type; (*Rinser inlet container presence*)
	IO_204DSF : IO_Digital_IN_Type; (*Container presence for filling valve opening*)
	IO_201DSF : IO_Digital_IN_Type; (*Filling valve 1 sensor*)
	IO_214DSF : IO_Digital_IN_Type; (*Head 1 Pulp Doser sensor //v999hema*)
	IO_204DSB : IO_Digital_IN_Type; (*Doser inlet container presence //v999hema*)
	IO_210CPF : IO_Valve_Type; (*Pulp Doser Pulp Valve Opening //v999hema*)
END_VAR
```

### IO_TNK.var
```iecst
(*MOTORS*)
VAR
	IO_PPF : ARRAY[MIN_CFG_VFD_PPx..MAX_CFG_VFD_PPx] OF IO_Motor_Type;
	IO_PPS : ARRAY[MIN_CFG_VFD_PPx..MAX_CFG_VFD_PPx] OF IO_Motor_Type;
END_VAR
(*DRIVERS*)
VAR
	IO_VFD_PPF : ARRAY[MIN_CFG_VFD_PPx..MAX_CFG_VFD_PPx] OF IO_PLK_Danfoss_Drive_Type;
	IO_VFD_PPS : ARRAY[MIN_CFG_VFD_PPx..MAX_CFG_VFD_PPx] OF IO_PLK_Danfoss_Drive_Type;
END_VAR
(*VALVES*)
VAR
	IO_AVF : ARRAY[MIN_CFG_AVx..MAX_CFG_AVx] OF IO_Valve_Type;
	IO_AVG : ARRAY[MIN_CFG_AVx..MAX_CFG_AVx] OF IO_Valve_Type;
	IO_AVS : ARRAY[MIN_CFG_AVx..MAX_CFG_AVx] OF IO_Valve_Type;
	IO_RVG : ARRAY[MIN_CFG_RVx..MAX_CFG_RVx] OF IO_Valve_Mod_Type;
	IO_RVF : ARRAY[MIN_CFG_RVx..MAX_CFG_RVx] OF IO_Valve_Mod_Type;
END_VAR
(*SENSORS*)
VAR
	IO_FSS : ARRAY[MIN_CFG_FSx..MAX_CFG_FSx] OF IO_Digital_IN_Type;
	IO_LSF : ARRAY[MIN_CFG_LSx..MAX_CFG_LSx] OF IO_Digital_IN_Type;
	IO_PSG : ARRAY[MIN_CFG_PSx..MAX_CFG_PSx] OF IO_Digital_IN_Type;
END_VAR
(*INSTRUMENTS*)
VAR
	IO_LTF : ARRAY[MIN_CFG_LTx..MAX_CFG_LTx] OF IO_Analog_IN_Type;
	IO_PTF : ARRAY[MIN_CFG_PTx..MAX_CFG_PTx] OF IO_Analog_IN_Type;
	IO_PTS : ARRAY[MIN_CFG_PTx..MAX_CFG_PTx] OF IO_Analog_IN_Type;
	IO_TTF : ARRAY[MIN_CFG_TTx..MAX_CFG_TTx] OF IO_Analog_IN_Type;
	IO_TTS : ARRAY[MIN_CFG_TTx..MAX_CFG_TTx] OF IO_Analog_IN_Type;
	IO_FTY : ARRAY[MIN_CFG_FTx..MAX_CFG_FTx] OF IO_Analog_IN_Type; (*V4.A.A.1.7.1*)
END_VAR
```

### IO_RNS.var
```iecst
VAR
	IO_202DSB : IO_Digital_IN_Type; (*GRIPPER RELEASED LIMIT SWITCH*)
	IO_206DSB : IO_Digital_IN_Type; (*NOB NOS OPENING CHECK SENSOR 2° TREAT.*)
	IO_205DSR : IO_Digital_IN_Type; (*GRIPPER "1" SENSOR*)
	IO_203PUB_1 : USINT;
	IO_203PUB_2 : USINT;
END_VAR
```

### IO_DOS.var
```iecst
VAR
	IO_209PUF_1 : USINT;
	IO_209PUF_2 : USINT;
	IO_209PUF_3 : USINT;
	IO_MMF : ARRAY[MIN_CFG_VFD_MMx..MAX_CFG_VFD_MMx] OF IO_MotorFC280_Type; (*//v999hema*)
	IO_VFD_MMF : ARRAY[MIN_CFG_VFD_MMx..MAX_CFG_VFD_MMx] OF IO_PLK_DanfossFC280_Drive_Type;
	IO_211CPF : IO_Valve_Type; (*Pulp Doser Cleaning Arm *)
	IO_PDO_YV65 : IO_Valve_Type; (*Pulp Doser Diaphram Pump PPJ203*)
	IO_210DSX : IO_Digital_IN_Type; (*Pulp Doser Arm in Cleaning Position*)
	IO_211DSX : IO_Digital_IN_Type; (*Pulp Doser Arm in Production Position*)
	IO_215DSF : IO_Digital_IN_Type; (*Pulp Doser HDP Up Limit Switch*)
	IO_216DSF : IO_Digital_IN_Type; (*Pulp Doser LDP Up Limit Switch*)
	IO_212DSF : IO_Digital_IN_Type; (*Pulp Doser Maximun Volume sensor *)
	IO_213DSF : IO_Digital_IN_Type; (*Pulp Doser Minimum Volume sensor *)
	IO_217DSF : IO_Digital_IN_Type; (*Pulp Doser LDP Down Limit Switch*)
	IO_DOS_OverloadOk : IO_Digital_IN_Type;
	IO_210PTF : IO_Digital_IN_Type;
	IO_205MEF : IO_Analog_IN_Type; (*Doser Pulp Volume HDP *)
	IO_206MEF : IO_Analog_IN_Type; (*Doser Pulp Volume LDP *)
END_VAR
```

### IO_C.var
```iecst
(*MOTORS*)
VAR
	IO_PPC : ARRAY[MIN_CFG_VFD_PPC..MAX_CFG_VFD_PPC] OF IO_Motor_Type;
END_VAR
(*DRIVERS*)
VAR
	IO_VFD_PPC : ARRAY[MIN_CFG_VFD_PPC..MAX_CFG_VFD_PPC] OF IO_PLK_Danfoss_Drive_Type;
END_VAR
(*VALVES*)
VAR
	IO_AVC : ARRAY[MIN_CFG_AVC..MAX_CFG_AVC] OF IO_Valve_Type;
	IO_HVC : ARRAY[MIN_CFG_HVC..MAX_CFG_HVC] OF IO_Valve_Type;
END_VAR
(*SENSORS*)
VAR
	IO_FSC : ARRAY[MIN_CFG_FSC..MAX_CFG_FSC] OF IO_Digital_IN_Type;
	IO_LSC : ARRAY[MIN_CFG_LSC..MAX_CFG_LSC] OF IO_Digital_IN_Type;
	IO_HSC : ARRAY[MIN_CFG_HSC..MAX_CFG_HSC] OF IO_Digital_IN_Type;
	IO_PSC : ARRAY[MIN_CFG_PSC..MAX_CFG_PSC] OF IO_Digital_IN_Type;
END_VAR
(*INSTRUMENTS*)
VAR
	IO_FTC : ARRAY[MIN_CFG_FTC..MAX_CFG_FTC] OF IO_Analog_IN_Type;
	IO_TTC : ARRAY[MIN_CFG_TTx..MAX_CFG_TTx] OF IO_Analog_IN_Type;
	IO_CTC : ARRAY[MIN_CFG_CTC..MAX_CFG_CTC] OF IO_Analog_IN_Type;
	IO_PTC : ARRAY[MIN_CFG_PTC..MAX_CFG_PTC] OF IO_Analog_IN_Type;
	IO_QTC : ARRAY[MIN_CFG_QTC..MAX_CFG_QTC] OF IO_Analog_IN_Type;
END_VAR
(*MODULATING VALVES*)
VAR
	IO_RVC : ARRAY[MIN_CFG_RVC..MAX_CFG_RVC] OF IO_Valve_Mod_Type; (*V4.A.A.1.7.1*)
END_VAR
```

### IO_COP.var
```iecst
VAR
	IO_201PUX_1 : USINT;
	IO_201PUX_2 : USINT;
	IO_201PUX_3 : USINT;
	IO_201PUE_1 : USINT;
	IO_201PUE_2 : USINT;
	IO_201PUE_3 : USINT;
	IO_201PUF_1 : USINT;
	IO_201PUF_2 : USINT;
	IO_202PUF_1 : USINT;
	IO_202PUF_2 : USINT;
	IO_PB_COP_FoamingGunStop : PB_Type;
	IO_PB_COP_FoamingGunRinse : PB_Type;
	IO_PB_COP_FoamingGunP1 : PB_Type;
	IO_PB_COP_FoamingGunP2 : PB_Type;
	IO_PB_COP_FoamingGunP3 : PB_Type;
END_VAR
```

### IO_B.var
```iecst
(*MOTORS*)
VAR
	IO_PPB : ARRAY[MIN_CFG_VFD_PPx..MAX_CFG_VFD_PPx] OF IO_Motor_Type;
END_VAR
(*DRIVERS*)
VAR
	IO_VFD_PPB : ARRAY[MIN_CFG_VFD_PPx..MAX_CFG_VFD_PPx] OF IO_PLK_DanfossFC280_Drive_Type;
END_VAR
(*VALVES*)
VAR
	IO_AVB : ARRAY[MIN_CFG_AVx..MAX_CFG_AVx] OF IO_Valve_Type;
	IO_HVB : ARRAY[MIN_CFG_HVx..MAX_CFG_HVx] OF IO_Valve_Type; (*V4.A.A.1.6.12*)
	IO_EVB : ARRAY[MIN_CFG_EVx..MAX_CFG_EVx] OF IO_Valve_Type; (*v1.7.4*)
	IO_206CPB : IO_Valve_Type; (*Moovable Spray Control  V4.A.A.1.7.0*)
	IO_296CPB : IO_Valve_Type; (*Moovable Cam ByPass Outlet Starwheel V4.A.A.1.7.0*)
	IO_297CPB : IO_Valve_Type; (*Moovable Cam ByPass Inlet Starwheel V4.A.A.1.7.0*)
	IO_298CPB : IO_Valve_Type; (*Moovable ByPass Starwheel Outlet Cam V4.A.A.1.7.0*)
	IO_299CPB : IO_Valve_Type; (*Moovable ByPass Starwheel Inlet Cam V4.A.A.1.7.0*)
END_VAR
(*SENSORS*)
VAR
	IO_FSB : ARRAY[MIN_CFG_FSx..MAX_CFG_FSx] OF IO_Digital_IN_Type;
	IO_LSB : ARRAY[MIN_CFG_LSx..MAX_CFG_LSx] OF IO_Digital_IN_Type;
	IO_HSB : ARRAY[MIN_CFG_HSx..MAX_CFG_HSx] OF IO_Digital_IN_Type; (*V4.A.A.1.6.12*)
	IO_PSB : ARRAY[MIN_CFG_PSx..MAX_CFG_PSx] OF IO_Digital_IN_Type; (*V4.A.A.1.7.0*)
	IO_QSB : ARRAY[MIN_CFG_QSx..MAX_CFG_QSx] OF IO_Digital_IN_Type; (*v1.7.4*)
	IO_298DSB : IO_Digital_IN_Type; (*V4.A.A.1.7.0*)
	IO_299DSB : IO_Digital_IN_Type; (*V4.A.A.1.7.0*)
END_VAR
(*INSTRUMENTS*)
VAR
	IO_FTB : ARRAY[MIN_CFG_FTx..MAX_CFG_FTx] OF IO_Analog_IN_Type; (*v1.7.4*)
	IO_TTB : ARRAY[MIN_CFG_TTx..MAX_CFG_TTx] OF IO_Analog_IN_Type;
	IO_CTB : ARRAY[MIN_CFG_CTx..MAX_CFG_CTx] OF IO_Analog_IN_Type;
	IO_PTB : ARRAY[MIN_CFG_PTx..MAX_CFG_PTx] OF IO_Analog_IN_Type; (*v1.7.4*)
	IO_LTB : ARRAY[MIN_CFG_LTx..MAX_CFG_LTx] OF IO_Analog_IN_Type; (*v1.7.4*)
	IO_QTB : ARRAY[MIN_CFG_QTx..MAX_CFG_QTx] OF IO_Analog_IN_Type; (*v1.7.4*)
END_VAR
(*MODULATING VALVES*)
VAR
	IO_RVB : ARRAY[MIN_CFG_RVx..MAX_CFG_RVx] OF IO_Valve_Mod_Type; (*V4.A.A.1.7.1*)
END_VAR
```

### IO_E.var
```iecst
(*MOTORS*)
VAR
	IO_PPE : ARRAY[MIN_CFG_VFD_PPx..MAX_CFG_VFD_PPx] OF IO_Motor_Type;
END_VAR
(*DRIVERS*)
VAR
	IO_VFD_PPE : ARRAY[MIN_CFG_VFD_PPx..MAX_CFG_VFD_PPx] OF IO_PLK_Danfoss_Drive_Type;
END_VAR
(*VALVES*)
VAR
	IO_AVE : ARRAY[MIN_CFG_AVx..MAX_CFG_AVx] OF IO_Valve_Type;
	IO_HVE : ARRAY[MIN_CFG_HVx..MAX_CFG_HVx] OF IO_Valve_Type; (*V4.A.A.1.6.12*)
END_VAR
(*SENSORS*)
VAR
	IO_FSE : ARRAY[MIN_CFG_FSx..MAX_CFG_FSx] OF IO_Digital_IN_Type;
	IO_LSE : ARRAY[MIN_CFG_LSx..MAX_CFG_LSx] OF IO_Digital_IN_Type;
	IO_PSE : ARRAY[MIN_CFG_PSx..MAX_CFG_PSx] OF IO_Digital_IN_Type;
END_VAR
(*INSTRUMENTS*)
VAR
	IO_FTE : ARRAY[MIN_CFG_FTx..MAX_CFG_FTx] OF IO_Analog_IN_Type;(*Master nuovo*)
	IO_LTE : ARRAY[MIN_CFG_LTx..MAX_CFG_LTx] OF IO_Analog_IN_Type;
	IO_PTE : ARRAY[MIN_CFG_PTx..MAX_CFG_PTx] OF IO_Analog_IN_Type;
	IO_AVEOCTET : ARRAY[0..1] OF USINT;
	IO_TTE : ARRAY[MIN_CFG_TTx..MAX_CFG_TTx] OF IO_Analog_IN_Type;
	IO_HSE : ARRAY[MIN_CFG_HSx..MAX_CFG_HSx] OF IO_Digital_IN_Type; (*V4.A.A.1.6.12*)
END_VAR
```

### IO_X.var
```iecst
(*MOTORS*)
VAR
	IO_PPX : ARRAY[MIN_CFG_VFD_PPx..MAX_CFG_VFD_PPx] OF IO_MotorFC280_Type;
END_VAR
(*DRIVERS*)
VAR
	IO_VFD_PPX : ARRAY[MIN_CFG_VFD_PPx..MAX_CFG_VFD_PPx] OF IO_PLK_DanfossFC280_Drive_Type;
END_VAR
(*VALVES*)
VAR
	IO_AVX : ARRAY[MIN_CFG_AVx..MAX_CFG_AVx] OF IO_Valve_Type;
END_VAR
(*SENSORS*)
VAR
	IO_FSX : ARRAY[MIN_CFG_FSx..MAX_CFG_FSx] OF IO_Digital_IN_Type;
	IO_LSX : ARRAY[MIN_CFG_LSx..MAX_CFG_LSx] OF IO_Digital_IN_Type;
	IO_TSX : ARRAY[MIN_CFG_TSx..MAX_CFG_TSx] OF IO_Digital_IN_Type;
	IO_PSX : ARRAY[MIN_CFG_PSx..MAX_CFG_PSx] OF IO_Digital_IN_Type;
END_VAR
(*INSTRUMENTS*)
VAR
	IO_PTX : ARRAY[MIN_CFG_PTx..MAX_CFG_PTx] OF IO_Analog_IN_Type;
END_VAR
```

### IO_Types.typ
```iecst
TYPE
	IO_MotionFanMachine_Type : 	STRUCT
		Filler : IO_MotionFanFiller_Type;
		Seamer : IO_MotionFanOutlet_Type;
	END_STRUCT;
	IO_MotionFanFiller_Type : 	STRUCT
		Main : IO_MotionFan_Type;
		In1 : IO_MotionFan_Type;
		In2 : IO_MotionFan_Type;
		In3 : IO_MotionFan_Type;
		In4 : IO_MotionFan_Type;
		In5 : IO_MotionFan_Type;
		In6 : IO_MotionFan_Type;
		In7 : IO_MotionFan_Type;
		In8 : IO_MotionFan_Type;
		In9 : IO_MotionFan_Type;
		In10 : IO_MotionFan_Type;
		Out1 : IO_MotionFan_Type;
		Out2 : IO_MotionFan_Type;
		Out3 : IO_MotionFan_Type;
		Out4 : IO_MotionFan_Type;
		Out5 : IO_MotionFan_Type;
	END_STRUCT;
	IO_MotionFanOutlet_Type : 	STRUCT
		Main : IO_MotionFan_Type;
	END_STRUCT;
	IO_Dmc_Type : 	STRUCT
		InsertionSensor : IO_Digital_IN_Type;
		InsertionPiston : IO_Valve_Type; (*Open = Inserction (Back)
Close = Disinserction (Forward)*)
	END_STRUCT;
	IO_OPS_Door_Type : 	STRUCT
		DI_Diagnostic : BOOL;
	END_STRUCT;
	IO_OPS_Zone_Type : 	STRUCT
		DO_GreenLight : BOOL;
		DO_RedLight : BOOL;
		DI_ConfinementAck : BOOL;
	END_STRUCT;
	IO_OPS_JOG_Type : 	STRUCT
		DI_Plugged : BOOL;
	END_STRUCT;
	IO_Cooling_Type : 	STRUCT
		MaxTemperature : BOOL; (*1.63 tolta inizializzazione variabile*)
		Overload : BOOL := TRUE;
	END_STRUCT;
	PO_Safety_Type : 	STRUCT  (*V4.A.A.1.6.13*)
		PB_Reset : BOOL; (*Push Button Command: Reset Push Button*)
		Production : BOOL; (*Machine on Production Running (the Product Inlet Valves stay Open with Doors Unlocked)*)
		PB_ResetBkInRoom : BOOL; (*Push Button Command: Room Door Inlet Reset Push Button*)
		PB_ResetBkOutRoom : BOOL; (*Push Button Command: Room Door Outlet Reset Push Button*)
		PB_ResetFwRoom : BOOL; (*Push Button Command: Room Door Outlet Reset Push Button*)
		BF_CoupledBF : BOOL; (*Combi Blower: Blower+Filler Coupled*)
		SSC_CoupledBlower : BOOL; (*SuperCombi BLF/BAF: Blower+Labeler / Blower+Actis Coupled//V4.A.A.1.6.10c*)
		SSC_CoupledFiller : BOOL; (*SuperCombi BLF/BAF: Labeler+Filler / Actis+Filler Coupled//V4.A.A.1.6.10c*)
		SSC_BF_BlowerAutoMode : BOOL; (*SuperCombi BLF/BAF ; Combi Blower: Blower on Automatic Mode//V4.A.A.1.6.10c*)
		SSC_LabActAutoMode : BOOL; (*SuperCombi BLF/BAF: Labeler/Actis on Automatic Mode//V4.A.A.1.6.10c*)
		SS_OP_FlrRelease : BOOL; (*Selector Switch Command: All Filler Door Release Command from HMI*)
		ReleaseEnable : BOOL; (*Filler Doors Release Enable Condition*)
		KeyJogReady : BOOL; (*JOG Enable Key: Inserted and Ready*)
		KeyJogWrong : BOOL; (*JOG Enable Key: Inserted but Wrong code*)
		BOOL114 : BOOL;
		BOOL115 : BOOL;
		BOOL116 : BOOL;
		BOOL117 : BOOL;
		HMI_UnlockSelector : BOOL; (*HMI Operator Protection Unlock Command (Selector Switch)V4.A.A.1.6.9*)
		HMI_LockSelector : BOOL; (*V4.A.A.1.6.9*)
		OP_BlwTrUnlockRequest : BOOL; (*Blower Transfer Doors Unlock Request*)
		OP_Lab_ActTrUnlockReq : BOOL; (*Super Combi BLF / BAF: Labeler / Actis Transfer Doors Unlock Requested//V4.A.A.1.6.10c*)
		BOOL122 : BOOL;
		BOOL123 : BOOL;
		BOOL124 : BOOL;
		CapArol_HighCommand : BOOL; (*Capper Arol: Buffer on High Positioning Command*)
		BOOL126 : BOOL;
		BOOL127 : BOOL;
		BOOL128 : BOOL;
		BOOL129 : BOOL;
		GeneralAirIn : BOOL; (*From SKID - 201PSG Inlet General Air Pressure: > 6.0 Bar = TRUE*)
		GeneralAirOut : BOOL; (*From SKID - Outlet General Air Valve 203EVG Opened*)
		BOOL132 : BOOL;
		BOOL133 : BOOL;
		BOOL134 : BOOL;
		HVB297 : BOOL; (*Sampling Valve Open Requested Command V4.A.A.1.6.10c*)
		BOOL136 : BOOL;
		BOOL137 : BOOL;
		BOOL138 : BOOL;
		BOOL139 : BOOL;
		BOOL142 : BOOL;
		BOOL143 : BOOL;
		BOOL144 : BOOL;
		BOOL145 : BOOL;
		BOOL146 : BOOL;
		BOOL147 : BOOL;
		BOOL148 : BOOL;
		FillerLiftRequ : BOOL; (*Filler Lifting enable request*)
		OpFwUnlock : BOOL; (*Operator Forward Door Lock-Unlock push Button*)
		OpBkInUnlock : BOOL; (*Operator Backward In Door Lock-Unlock push Button*)
		OpBkOutUnlock : BOOL; (*Operator Backward Out Door Lock-Unlock push Button*)
		OpTrFwUnlock : BOOL; (*Operator Trasfer In Door Lock-Unlock push Button*)
		OpTrBkUnlock : BOOL; (*Operator Trasfer Out Door Lock-Unlock push Button*)
	END_STRUCT;
	PI_Safety_Type : 	STRUCT  (*V4.A.A.1.6.13*)
		OP_ConfirmPB : BOOL; (*OP Safety Flag: Area Doors Opened Confirm Push Button - Green Lamp V4.A.A.1.6.9*)
		OPFw_ConfirmRequest : BOOL; (*OP Filler Forward Safety Flag: Area Doors Opened Confirm Request - Red Lamp*)
		OPBkIn_ConfirmRequest : BOOL; (*OP Filler Backward Inlet Safety Flag: Area Doors Opened Confirm Request - Red Lamp*)
		OPBkOut_ConfirmRequest : BOOL; (*OP Filler Backward Outlet Safety Flag: Area Doors Opened Confirm Request - Red Lamp*)
		OPTrFw_ConfirmRequest : BOOL; (*OP Filler Transfer Forwrd Safety Flag: Area Doors Opened Confirm Request - Red Lamp*)
		OPTrBk_ConfirmRequest : BOOL; (*OP Filler Transfer Backward Safety Flag: Area Doors Opened Confirm Request - Red Lamp*)
		OPRnBkIn_ConfirmRequest : BOOL; (*OP Rinser Backward Inlet Safety Flag: Area Doors Opened Confirm Request - Red Lamp*)
		OPRnBkOut_ConfirmRequest : BOOL; (*OP Rinser Backward Outlet Safety Flag: Area Doors Opened Confirm Request - Red Lamp*)
		BOOL009 : BOOL;
		OPFw_Jog : BOOL; (*OP Forward Safety Flag: Jog Selected*)
		OPBkIn_Jog : BOOL; (*OP Backward Inlet Safety Flag: Jog Selected*)
		OPBkOut_Jog : BOOL; (*OP Backward Outlet Safety Flag: Jog Selected*)
		OPTrFw_Jog : BOOL; (*OP Transfer Forward Safety Flag: Jog Selected*)
		OPMnOut_Jog : BOOL; (*OP Capper Platform Safety Flag: Jog Selected*)
		OPRnBkIn_Jog : BOOL; (*OP Rinser Backward Inlet Safety Flag: Jog Selected*)
		OPRnBkOut_Jog : BOOL; (*OP Rinser Backward Outlet Safety Flag: Jog Selected //V4.A.A.1.6.10c*)
		OPFwEx_Jog : BOOL; (*OP Forward External Safety Flag: Jog Selected //vrma 106*)
		OPFwEx_JogError : BOOL; (*OP Forward External Safety Flag: Jog Selected Fault vrma106*)
		BOOL019 : BOOL;
		SS_LockOutOff : BOOL; (*V4.A.A.1.7.1*)
		SS_LockOutError : BOOL; (*V4.A.A.1.7.1*)
		SS_JogKeyOff : BOOL; (*Jog with Door Opened Enable Key: Selector on Off Position V4.A.A.1.7.1*)
		SS_JogKeyError : BOOL; (*Jog with Door Opened Enable Key: Selector on Fault V4.A.A.1.7.1*)
		GateConveyorClosed : BOOL; (*OP Filler Safety Flag: Outlet Conveyor Gate Closed*)
		GateConveyorShCirc : BOOL; (*OP Filler Safety Flag: Outlet Conveyor Gate Short Circuit*)
		OPTrGateClosed : BOOL; (*OP Transfer Gate Safety Flag: Gate Closed (Isolation Door Installed)*)
		OPTrGateShCirc : BOOL; (*OP Transfer Gate Safety Flag: Gate Short Circuit (Isolation Door)*)
		BOOL028 : BOOL;
		BOOL029 : BOOL;
		BOOL030 : BOOL;
		BOOL031 : BOOL;
		BOOL032 : BOOL;
		BOOL033 : BOOL;
		BOOL034 : BOOL;
		BOOL035 : BOOL;
		BOOL036 : BOOL;
		OP_ClosedRnsPw : BOOL; (*Operator Protection Safety Flag: Operator Protection Closed Rinser Power ON (Delay)V4.A.A.1.6.10c*)
		OP_ClosedRnsPwFault : BOOL; (*Operator Protection Safety Flag: Operator Protection Closed Rinser Power Fault V4.A.A.1.6.10c*)
		OP_UnlockOpened : BOOL; (*Operator Protection Safety Flag: Operator Protection Unlocked/Opened (HMI Selector=Orange)V4.A.A.1.6.9*)
		OP_CLOSED : BOOL; (*Operator Protection Safety Flag: OPERATOR PROTECTION CLOSED*)
		OP_ExtTrCLOSED : BOOL; (*Operator Protection Safety Flag: External Machine Transfer Doors Closed*)
		OP_ClosedFlrPw : BOOL; (*Operator Protection Safety Flag: Operator Protection Closed Rinser Power ON (Delay) V4.A.A.1.6.10c*)
		OP_ClosedFlrPwFault : BOOL; (*Operator Protection Safety Flag: Operator Protection Closed Filler Power Fault V4.A.A.1.6.10c*)
		BOOL044 : BOOL;
		OP_RELEASE_REQUEST : BOOL; (*Operator Protection Safety Flag: RELEASE REQUEST - MACHINE STOP*)
		OP_RELEASE_Fault : BOOL; (*Operator Protection Safety Flag: RELEASE CIRCUIT FAULT*)
		OP_TransferReleaseRequest : BOOL; (*Operator Protection Safety Flag: Transfer Area Release Request - Sent to Near Machine V4.A.A.1.6.10c*)
		BOOL048 : BOOL;
		BOOL049 : BOOL;
		EMERGENCY_ON : BOOL; (*EMERGENCY CIRCUIT READY*)
		EMERGENCY_CircuitFault : BOOL; (*EMERGENCY CIRCUIT FAULT*)
		EMERGENCY_FILLER : BOOL; (*EMERGENCY FILLER CIRCUIT READY*)
		EMERGENCY_BLOWER : BOOL; (*EMERGENCY BLOWER CIRCUIT READY*)
		EMERGENCY_BLOWER_Fault : BOOL; (*EMERGENCY BLOWER CIRCUIT Feed-Back Fault*)
		EMERGENCY_LABELER : BOOL; (*EMERGENCY LABELER CIRCUIT READY*)
		EMERGENCY_LABELER_Fault : BOOL; (*EMERGENCY LABELER CIRCUIT Feed-back Fault*)
		EmgSkidFault : BOOL; (*Emergency Skid Feed-Back Circuit FAULT*)
		FillerLiftPw : BOOL; (*Master nuovo*)
		FillerLiftPwFault : BOOL; (*Master nuovo*)
		SelMode_Auto : BOOL; (*Mode Selection: Automatic*)
		SelMode_JOG : BOOL; (*Mode Selection: JOG*)
		SelMode_Setting : BOOL; (*Mode Selection: Setting*)
		SelMode_Error : BOOL; (*Mode Selection: Selection Error "JOG Selected from External Machine"*)
		JOG_StopPB : BOOL; (*STOP Push Button on JOG Pressed*)
		JOG_Control_Error : BOOL; (*Jog Safety Flag: JOG Connection Error -Too much Jog Inserted*)
		Selector_Auto : BOOL; (*Selector mode position: Automatic*)
		SelModeAutoError : BOOL; (*Mode Selection: Automatic Error (JOG Enable Key Inserted)*)
		SelModeChange : BOOL; (*Mode Selection: Mode Change, machine Stopped requested*)
		BOOL069 : BOOL;
		DriveEnable : BOOL; (*Emergency + (Operator Protection * JOG) Drive Enabled*)
		JOG_Run : BOOL; (*Jog Safety Flag: JOG Run Command*)
		DriveSafeOFFTimeOut : BOOL; (*Drive Control: Machine Safe OFF Time Out*)
		DriveStopTimeOut : BOOL; (*Drive Control: Machine Stop Time Out*)
		JOG_SpeedError : BOOL; (*Filler JOG Speed Fault*)
		BOOL077 : BOOL;
		BOOL078 : BOOL;
		BOOL079 : BOOL;
		AirReady : BOOL; (*General Air ON: Ready*)
		AirCloseOP : BOOL; (*General Air OFF: Close the Operator Guard to Have Pressure*)
		ProcessValvesFault : BOOL; (*Filler Process Valves Feed-Back Fault*)
		CopValvesFault : BOOL; (*Filler Cop/Washing Valves Feed-Back Fault*)
		VbsValvesFault : BOOL; (*Nitrodoser valves Feed-Back fauòlt*)
		BOOL085 : BOOL;
		BOOL086 : BOOL;
		BOOL087 : BOOL;
		BOOL088 : BOOL;
		BOOL089 : BOOL;
		BOOL090 : BOOL;
		EMERGENCY_VBS : BOOL; (*EMERGENCY VBS READY //CANCELED in Safety document 40v0*)
		EmgVbsPressed : BOOL; (*Emergency Vbs Pressed //CANCELED in Safety document 40v0*)
		EmgVbsShc : BOOL; (*Emergency Vbs Fault //CANCELED in Safety document 40v0*)
		EMERGENCY_CONVEYOR : BOOL; (*EMERGENCY CONVEYOR READY*)
		EmgConveyorPressed : BOOL; (*Emergency Conveyor Pressed*)
		EmgConveyorSch : BOOL; (*Emergency Conveyor Fault*)
		CapBufOP_CLOSED : BOOL; (*Capper Buffer: Buffer Area Closed*)
		CapBuf2OP_CLOSED : BOOL; (*Capper Buffer 2 /Hopper External 2: Buffer Area Closed V4.A.A.1.6.10c*)
		CapBufOP1_Opened : BOOL; (*Capper Buffer: Buffer Door 1 Opened*)
		CapBufOP2_Opened : BOOL; (*Capper Buffer: Buffer Door 2 Opened*)
		CapBufOP1_Sch : BOOL; (*Capper Buffer: Buffer Door 1 Short Circuit  Safety*)
		CapBufOP2_Sch : BOOL; (*Capper Buffer: Buffer Door 2 Shor Circuit Safety*)
		BOOLext0007 : BOOL;
		CapBufEx_DriveEnable : BOOL; (*Capper Buffer/Hopper External: Drive Enable V4.A.A.1.6.10c*)
		CapMotionEnable : BOOL; (*Capper Motion Head Rotation: Motion Enable (Arol Equatorque/Zalkin) V4.A.A.1.6.10c*)
		BOOLext0010 : BOOL;
		BOOLext0011 : BOOL;
		BOOLext0012 : BOOL;
		CapBuf2OP1_Opened : BOOL; (*Capper Buffer/Hopper External: Buffer Door 1 Opened V4.A.A.1.6.10c*)
		CapBuf2OP2_Opened : BOOL; (*Capper Buffer/Hopper External: Buffer Door 2 Opened V4.A.A.1.6.10c*)
		CapBuf2OP1_Sch : BOOL; (*Capper Buffer/Hopper External: Buffer Door 1 Short Circuit  Safety V4.A.A.1.6.10c*)
		CapBuf2OP2_Sch : BOOL; (*Capper Buffer/Hopper External: Buffer Door 2 Shor Circuit Safety V4.A.A.1.6.10c*)
		BOOLext0017 : BOOL;
		BOOLext0018 : BOOL;
		BOOLext0019 : BOOL;
		CapArolPosReady : BOOL; (*Arol Capper Buffer: Position Ready for Doors Unlock*)
		CapArolPosFault : BOOL; (*Arol Capper Buffer: Position Fault*)
		CapArolHighFault : BOOL; (*Arol Capper Buffer: High Position Feed-Back Fault*)
		CapArolBlockedFault : BOOL; (*Arol Capper Buffer: Blocked Position Feed-Back Fault*)
		BOOLext0024 : BOOL;
		CapExtr1Op_Opened : BOOL; (*Cap Extractor 1: Door Opened*)
		CapExtr1Op_Shc : BOOL; (*Cap Extractor 1: Door Short Circuit Safety*)
		CapExtr2Op_Opened : BOOL; (*Cap Extractor 2: Door Opened*)
		CapExtr2Op_Shc : BOOL; (*Cap Extractor 2: Door Short Circuit Safety*)
		BOOLext0029 : BOOL;
		MO_BLO_BaseTest : BOOL; (*Machine Option: BLO Base Machine Test -> "SafeMachineOption00" (on Test = SAFETRUE)V4.A.A.1.6.10c*)
		BOOLext0031 : BOOL;
		MO_BLO_CnfError : BOOL; (*Machine Option: BLO Configuration Error -> Emergency Stop (SefeMachineOption00 = SAFETRUE with Hardware present) V4.A.A.1.6.10c*)
		OPFw_AreaState_AreaError : UINT; (*OP Forward (Zone 1+11): Area State / Area Error*)
		OPBkIn_AreaState_AreaError : UINT; (*OP Backward Inlet (Zone 2+12): Area State / Area Error*)
		OPBkOut_AreaState_AreaError : UINT; (*OP Backward Outlet (Zone 3+13): Area State / Area Error*)
		OPTrFw_AreaState_AreaError : UINT; (*OP Transfer Forward (Zone 4): Area State / Area Error*)
		OPTrBk_AreaState_AreaError : UINT; (*OP Transfer Backward (Zone 5): Area State / Area Error*)
		OPTrFw_TrBk_StateError : UINT; (*OP Transfer Forward/Transfer Backward: Doors State/Doors Error*)
		OPMnIn_AreaState_AreaError : UINT; (*OP Maintenance Inlet (Zone 7): Area State / Area Error*)
		OPMnOut_AreaState_AreaError : UINT; (*OP Maintenance Outlet (Zone 8) Area State / Area Error*)
		OPMnIn_MnOut_StateError : UINT; (*OP Maintenance Inlet/Maintenance Outlet: Doors State/Doors Error*)
		OPRnBkIn_AreaState_AreaErr : UINT; (*OP Rinser Backward Inlet (Zone16): Area State / Area Error*)
		OPRnBkIn_OpenedConfirm : UINT; (*OP Rinser Backward Inlet (Zone 16): Doors 1-:-8 Opened/Confirm*)
		OPRnBkIn_Lock1oo2LockSafety : UINT; (*OP Rinser Backward Inlet (Zone 16): Doors 1-:-8 Lock_1oo2/Lock_Safety*)
		OPRnBkIn_UnlockedShcError : UINT; (*OP Rinser Backward Inlet (Zone 16): Doors 1-:-8 Unlocked/Short Circuit*)
		OPRnBkOut_AreaState_AreaErr : UINT; (*OP Rinser Backward Outlet (Zone 17): Area State / Area Error*)
		OPRnBkOut_OpenedConfirm : UINT; (*OP Rinser Backward Outlet (Zone 17): Doors 1-:-8 Opened/Confirm*)
		OPRnBkOut_Lock1oo2LockSaf : UINT; (*OP Rinser Backward Outlet (Zone 17): Doors 1-:-8 Lock_1oo2/Lock_Safety*)
		OPRnBkOut_UnlockedShcError : UINT; (*OP Rinser Backward Outlet (Zone 17): Doors 1-:-8 Unlocked/Short Circuit*)
		OPRnMnOut_AreaState_AreaErr : UINT; (*OP Rinser Maintenance Outlet (Zone 18): Area State / Area Error*)
		OPRnMnIn_MnOut_StateError : UINT; (*OP Rinser Maintenance Inlet/Maintenance Outlet: Doors State/Doors Error*)
		UINT020 : UINT;
		UINT021 : UINT;
		UINT022 : UINT;
		EmgPB_Press : UINT; (*Filler Emergency Pus Button 1-:-8 Pressed*)
		EmgPB_Shc : UINT; (*Filler Emergency Pus Button 1-:-8 Short Circuit*)
		EmgDriveFault : UINT; (*Emergency Circuit Drive Safe OFF Feed Back Fault*)
		EmgOpDriveFault : UINT; (*Emergency + Operator Protection Circuit Drive Safe OFF Feed Back Fault*)
		EmgOpJogDriveFault : UINT; (*Emergency + (Operator Protection * Jog) Circuit Drive Safe OFF Feed Back Fault*)
		OPValveFault : UINT; (*Operator Protection Circuit Valves Closed Feed Back Fault V4.A.A.1.7.0*)
		SwVer1 : UINT; (*Configuration: Software Version First/Second Digit V4.A.A.1.6.10c*)
		SwVer2 : UINT; (*Configuration: Software Version Third/Fourth Digit V4.A.A.1.6.10c*)
		OPFw_Opened_Confirm : UDINT; (*OP Forward: Zone 1 _ Zone 11: Doors Opened/Confirm*)
		OPFw_Lock1oo2_LockSafety : UDINT; (*OP Forward: Zone 1 _ Zone 11: Doors Lock_1oo2/Lock_Safety*)
		OPFw_Unlocked_ShcError : UDINT; (*OP Forward: Zone 1 _ Zone 11: Doors Unlocked/Short Circuit*)
		OPBkIn_Opened_Confirm : UDINT; (*OP Backward Inlet: Zone 2 _ Zone 12: Doors Opened/Confirm*)
		OPBkIn_Lock1oo2_LockSafety : UDINT; (*OP Backward Inlet: Zone 2 _ Zone 12 Doors Lock_1oo2/Lock_Safety*)
		OPBkIn_Unlocked_ShcError : UDINT; (*OP Backward Inlet: Zone 2 _ Zone 12 Doors Unlocked/Short Circuit*)
		OPBkOut_Opened_Confirm : UDINT; (*OP Backward Outlet: Zone 3 _ Zone 13 Doors Opened/Confirm*)
		OPBkOut_Lock1oo2_LockSafety : UDINT; (*OP Backward Outlet: Zone 3 _ Zone 13 Doors Lock_1oo2/Lock_Safety*)
		OPBkOut_Unlocked_ShcError : UDINT; (*OP Backward Outlet: Zone 3 _ Zone 13 Doors Unlocked/Short Circuit*)
		OPPdBkIn_Opened_Confirm : UDINT; (*OP Pulp Doser Backward Inlet: Zone 21 _ Zone 22: Doors Opened/Confirm*)
		OPPdBkIn_Lock1oo2_LockSafety : UDINT; (*OP Pulp Doser Backward Inlet: Zone 21 _ Zone 22 Doors Lock_1oo2/Lock_Safety*)
		OPPdBkIn_Unlocked_ShcError : UDINT; (*OP Pulp Doser Backward Inlet: Zone 21 _ Zone 22 Doors Unlocked/Short Circuit*)
		UDINT013 : UDINT;
		CnfAreaPresent : UDINT; (*Operator Protection Zone Presence*)
	END_STRUCT;
	IO_SS3PModality_Type : 	STRUCT
		DI_Adjustement : BOOL; (*Adjustement*)
		DI_Auto : BOOL; (*Auto*)
		DI_Jog : BOOL; (*Jog*)
	END_STRUCT;
	IO_MCRaw_Type : 	STRUCT
		Input : IO_MCRawInput_Type;
		Output : IO_MCRawOutput_Type;
	END_STRUCT;
	IO_MCRawInput_Type : 	STRUCT
		MachineCommand : ARRAY[0..31]OF USINT;
		MachineReference : ARRAY[0..31]OF USINT;
		FillerCommandReference : ARRAY[0..31]OF USINT;
		PAR : ARRAY[0..127]OF USINT;
	END_STRUCT;
	IO_MCRawOutput_Type : 	STRUCT
		MachineAlarm : ARRAY[0..31]OF USINT;
		MachineStatus : ARRAY[0..31]OF USINT;
		FillerStatusAlarm : ARRAY[0..31]OF USINT;
	END_STRUCT;
	IO_SiriusStarter_Type : 	STRUCT  (*//V4.A.A.1.6.11*)
		DI_Fault : IO_Digital_IN_Type;
		DO_CW : BOOL;
		DO_CCW : BOOL;
	END_STRUCT;
	IO_ITC_Type : 	STRUCT
		CVO : IO_ITC_CVO_Type;
		VBC : IO_ITC_VBC_Type;
		FILTEC : IO_ITC_FCI_Type; (*v1.65*)
		STRATEC : IO_ITC_FCI_Type; (*v1.65*)
		PRESSCO : IO_ITC_FCI_Type; (*v1.65*)
		HEUFT : IO_ITC_FCI_Type; (*v1.65*)
		FTSYSTEM : IO_ITC_FCI_Type; (*v1.65*)
		SIS : IO_ITC_FCI_Type; (*v1.65*)
		COP : IO_ITC_COP_Type;
		UVL : IO_ITC_UVL_Type; (*v1.63*)
		CFD : IO_ITC_CFD_Type; (*V4.A.A.1.6.12*)
		SIKO : IO_ITC_SIKO_Type; (*V4.A.A.1.6.12*)
		DOS : IO_ITC_DOS_Type; (*V4.A.A.1.6.11*)
		CVI : IO_ITC_CVI_DP_Type; (*V4.A.A.1.6.14*)
		CFD2 : IO_ITC_CFD_Type; (*V4.A.A.1.7.1*)
		CDR : IO_ITC_CDR_Type; (*V4.A.A.1.7.1*)
	END_STRUCT;
	IO_ITC_UVL_Type : 	STRUCT
		In : UvlFlr_Type;
		Out : FlrUvl_Type;
	END_STRUCT;
	IO_ITC_CVO_Type : 	STRUCT
		In : CvoFlr_Type;
		Out : FlrCvo_Type;
	END_STRUCT;
	IO_ITC_VBC_Type : 	STRUCT
		In : VbcFlr_Type;
		Out : FlrVbc_Type;
	END_STRUCT;
	IO_ITC_FCI_Type : 	STRUCT
		In : FciFlr_Type;
		Out : FlrFci_Type;
	END_STRUCT;
	IO_ITC_COP_Type : 	STRUCT
		In : CopFlr_Type;
		Out : FlrCop_Type;
	END_STRUCT;
	IO_ITC_CFD_Type : 	STRUCT  (*V4.A.A.1.6.12*)
		In : CfdFlr_Type;
		Out : FlrCfd_Type;
	END_STRUCT;
	IO_ITC_DOS_Type : 	STRUCT  (*V4.A.A.1.6.11*)
		In : DosFlr_Type;
		Out : FlrDos_Type;
	END_STRUCT;
	IO_CSR_SCU_Type : 	STRUCT
		DI_OverloadOK : BOOL;
		DI_ContactorFBK : BOOL; (*Contactor Feed-Back *)
		DI_SafetyEnable : BOOL; (*Safety Enable from IOMapping*)
		DO_StorePosition : BOOL;
		DO_PowerON : BOOL;
		DO_Down : BOOL;
		DO_Up : BOOL;
		DI_Powered : BOOL; (*master nuovo*)
		DO_PowerOn : BOOL; (*Master nuovo*)
	END_STRUCT;
	IO_CPU_Type : 	STRUCT
		BatteryStatus : USINT; (*Battery status CPU (0 = battery low or missing, 1 = battery ok,)*)
		CoolingPlateTemperature : INT; (*Temperature cooling plate [1/10C] vrma*)
		Temperature : INT; (*Temperature CPU [1/10C] vrma*)
	END_STRUCT;
	IO_UPS_Type : 	STRUCT
		DI_BatteryReady : BOOL; (*True = UPS in alarm*)
		DI_Alarm : BOOL; (*True = Battery > 85%*)
		DI_MainPowerOn : BOOL := TRUE; (*True = Main power supply on*)
		DI_ModuleOk : BOOL;
		DO_HmiRestart : BOOL;
	END_STRUCT;
	IO_ITC_SIKO_Type : 	STRUCT  (* *) (* *) (*80*)
		In : SikoFlr_Type; (* *) (* *) (*82*)
		Out : FlrSiko_Type; (* *) (* *) (*81*)
	END_STRUCT;
	IO_ITC_CVI_DP_Type : 	STRUCT  (*V4.A.A.1.6.14*)
		In : ARRAY[0..9]OF USINT;
		Out : ARRAY[0..9]OF USINT;
	END_STRUCT;
	IO_ITC_CDR_Type : 	STRUCT  (*V4.A.A.1.7.0*)
		In : CdrFlr_Type;
		Out : FlrCdr_Type;
	END_STRUCT;
END_TYPE
```

### IO_BTC.var - not listed in the package file held
```iecst
VAR
	IO_BTC_UVL : ARRAY[200..201] OF IO_UVtronic_Type;
END_VAR
```

### Package Logical/00_AID/Modules - Global Modules variables

### AID_Global.typ
```iecst
(*AUXILIARY MEMORY*)

TYPE
	AID_Type : 	STRUCT
		DataOut : AID_DataOut_Type;
	END_STRUCT;
	AID_DataOut_Type : 	STRUCT
		Blink05Hz : BOOL;
		Blink1Hz : BOOL;
		Blink4Hz : BOOL;
		Blink2Hz : BOOL;
		Blink5Hz : BOOL; (*v1.7.5*)
		NetBlinkSlow : BOOL; (*Almost 1Hz*)
		NetBlinkFast : BOOL; (*Almost 4Hz*)
		Reset : BOOL;
		OperatorPresence : BOOL;
		OneContainerStopAlarm : BOOL; (*V4.A.A.1.6.13*)
		OneMachineStopAlarm : BOOL; (*V4.A.A.1.6.13*)
		ALR : ActionSum_Type;
		ProjectType : USINT;
	END_STRUCT;
END_TYPE
```

### RNS_Global.typ
```iecst
(*RINSER*)

TYPE
	RNS_Type : 	STRUCT  (*V4.A.A.1.7.0*)
		DataOut : RNS_DataOut_Type;
	END_STRUCT;
	RNS_DataOut_Type : 	STRUCT  (*V4.A.A.1.7.0*)
		Idle : BOOL;
		StepCountReq : BOOL;
		CipMode : BOOL;
		CipDrainMode : BOOL;
		RinseMode : BOOL;
		DrainMode : BOOL;
		ProdMode : BOOL;
		StartUp : BOOL;
		CopMode : BOOL;
		DeEnergization : BOOL;
		SystemTreatmentAlr : BOOL;
		SystemOnTreatment : BOOL;
		InsercionRequest : BOOL;
		ByPassRequest : BOOL;
		ControlContinousRequestWater : BOOL;
		ControlContinousRequestAir : BOOL;
		ControlInsercionRequestWater : BOOL;
		ControlInsercionRequestAir : BOOL;
		FixSpeedRequest : BOOL;
		ByPassed : BOOL;
		AxisDisableRequest : BOOL;
		ContainerStop : BOOL;
		CipDrainEnd : BOOL;
		InsrtcionDeviceRequest : BOOL;
		InsrtcionControlActive : BOOL;
		ContinousControlActive : BOOL;
		ProductRequest : BOOL;
		StepCounterRequest : BOOL;
		MachineStart : BOOL;
		MachineStop : BOOL;
		NoBottleNoSprayInsercion : BOOL; (*vrma test*)
		BottlesNotRinse : BOOL;
		CipDisableAxisReq : BOOL; (*//RnsDisable*)
		WaterFlow : REAL;
		Temperature : REAL;
		FixSpeedValue : REAL;
	END_STRUCT;
	RNS_NozzleData_Type : 	STRUCT  (*V4.A.A.1.7.0*)
		Visibility : BOOL;
		InsercionAir : RNS_Control_Type;
		InsercionWater : RNS_Control_Type;
		ContinousAir : RNS_Control_Type;
		ContinousWater : RNS_Control_Type;
		NozzleNumber : USINT;
	END_STRUCT;
	RNS_Control_Type : 	STRUCT  (*V4.A.A.1.7.0*)
		Active : BOOL;
		Alarm : BOOL;
		FailedCount : USINT;
	END_STRUCT;
END_TYPE
```

### CAP_Global.typ
```iecst
(*CAPPER*)

TYPE
	CAP_Config_Type : 	STRUCT
		ChannelA : BOOL;
		ChannelB : BOOL;
		ChannelC : BOOL;
		HeadRotationDir : BOOL;
		BufferSize : UINT;
		PickAndPlace : UINT;
		CamHeightPosition : USINT;
	END_STRUCT;
	CAP_Head_Type : 	STRUCT  (*v1.5*)
		HeadNr : UINT; (*Head Displayed on Row*)
		Data1 : UINT;
		Data2 : UINT;
		Totalizer00 : UINT;
		Totalizer01 : UINT;
		Totalizer02 : UINT;
		Totalizer03 : UINT;
		Totalizer04 : UINT;
		Totalizer05 : UINT;
		Totalizer06 : UINT;
		Totalizer07 : UINT;
		Bool00 : BOOL;
		Bool01 : BOOL;
		Bool02 : BOOL;
		Bool03 : BOOL;
		Bool04 : BOOL;
		Bool05 : BOOL;
		Bool06 : BOOL;
		Bool07 : BOOL;
		LineVisibility : BOOL;
	END_STRUCT;
	CAP_Mode_Type :
		(
		CAP_Idle,
		CAP_Production,
		CAP_ProductionReady,
		CAP_Emptying,
		CAP_EmptyingRunning,
		CAP_EmptyingDone,
		CAP_BufferLifting,
		CAP_BufferLiftingDone,
		CAP_BufferLowering,
		CAP_BufferLoweringDone,
		CAP_SizeChange,
		CAP_SizeChangeDone
		);
	CAP_SikoMode_Type :
		(
		SikoMbd_Idle,
		SikoMbd_ManualPositioningHoming,
		SikoMbd_ManualPositioning,
		SikoMbd_WriteParameterM171,
		SikoMbd_WriteParameterM172,
		SikoMbd_WriteParameterM173,
		SikoMbd_PosizioningTimeout,
		SikoMbd_AutoPositioning,
		SikoMbd_MachineEmptying
		);
	CAP_CamMode_Type :
		(
		CamSizeChange_Init,
		Cam_SizeChange_WaitOperator,
		Cam_SizeChange_WaitMachineStop,
		Cam_SizeChange_Unlock,
		Cam_SizeChange_Move,
		Cam_SizeChange_Lock,
		Cam_SizeChange_WaitOperatorOff,
		Cam_SizeChange_Done
		);
	CAP_BufferMode_Type :
		(
		Buffer_Idle,
		Buffer_StartUp,
		Buffer_StartUpFilling,
		Buffer_StartUpFillingTimeOut,
		Buffer_Production,
		Buffer_ProductionLowLevel,
		Buffer_EndProductionFilled,
		Buffer_EndProductionEmptying,
		Buffer_EmptyingRotationReverse,
		Buffer_MotorRotationStop,
		Buffer_Emptying,
		Buffer_EmptyingOpenGate,
		Buffer_EmptyingTimeOut,
		Buffer_EmptyingFW1,
		Buffer_EmptyingFW1TimeOut,
		Buffer_EmptyingFW2,
		Buffer_EmptyingFW2TimeOut,
		Buffer_EmptyingFWStopRotation,
		Buffer_EmptyingBW,
		Buffer_EmptyingBWStopRotation,
		Buffer_EmptyingFW3,
		Buffer_EmptyingDone,
		Buffer_MovingUp,
		Buffer_MovingUpRemoveBlock,
		Buffer_MovingUpLifting,
		Buffer_MovingUpInsertBlock,
		Buffer_MovingUpCompleted,
		Buffer_MovingUpLiftingError,
		Buffer_MovingUpBlockError,
		Buffer_MovingDown,
		Buffer_MovingDownWaitOperator,
		Buffer_MovingDownCheckCaps,
		Buffer_MovingDownLifting,
		Buffer_MovingDownRemoveBlock,
		Buffer_MovingDownLowering,
		Buffer_MovingDownInsertBlock,
		Buffer_MovingDownCompleted,
		Buffer_MovingDownLoweringError,
		Buffer_MovingDownLiftingError,
		Buffer_MovingDownBlockError,
		Buffer_SizeChangeInit,
		Buffer_SizeChangeGuideLift,
		Buffer_SizeChangeGuideLow,
		Buffer_SizeChangeGuideHigh,
		Buffer_SizeChangeGuideLower,
		Buffer_SizeChangeGuideUnlock,
		Buffer_SizeChangeGuideLock,
		Buffer_SizeChangeDone,
		Buffer_AdjustmentInit, (*//V4.A.A.1.6.11*)
		Buffer_AdjustmentPositionToZero, (*//V4.A.A.1.6.11*)
		Buffer_AdjustmentZeroToPosition, (*//V4.A.A.1.6.11*)
		Buffer_AdjustmentPositionReached, (*//V4.A.A.1.6.11*)
		Buffer_AdjustmentDone, (*//V4.A.A.1.6.11*)
		Buffer_AdjustmentFault (*//V4.A.A.1.6.12h*)
		);
	CAP_EquCalMode_Type :
		( (*//V4.A.A.1.6.12 Calibration Sequence*)
		Wait_Start, (*Wait For Calibration Start V4.A.A.1.6.12*)
		Reset_Data, (*Calibration Data Reset V4.A.A.1.6.12*)
		Empty1_SaveCurrent, (*Calibration 1 without Friction -Save Current V4.A.A.1.6.12*)
		Empty1_Done, (*Calibration 1 Done V4.A.A.1.6.12*)
		Empty2_SaveCurrent, (*Calibration 2 without Friction -Save Current V4.A.A.1.6.12*)
		Empty2_Done, (*Calibration 2 Done V4.A.A.1.6.12*)
		Empty3_SaveCurrent, (*Calibration 3 without Friction -Save Current V4.A.A.1.6.12*)
		Empty3_Done, (*Calibration 3 Done V4.A.A.1.6.12*)
		Wait_Friction, (*Wait For Friction Installation V4.A.A.1.6.12*)
		Friction1_SaveCurrent, (*Calibration 1 with Friction -Save Current V4.A.A.1.6.12*)
		Friction1_Done, (*Calibration 1 with Friction Done V4.A.A.1.6.12*)
		Friction2_SaveCurrent, (*Calibration 2 with Friction -Save Current V4.A.A.1.6.12*)
		Friction2_Done, (*Calibration 2 with Friction  Done V4.A.A.1.6.12*)
		Friction3_SaveCurrent, (*Calibration 3 with Friction -Save Current V4.A.A.1.6.12*)
		Friction3_Done, (*Calibration 3 with Friction  Done V4.A.A.1.6.12*)
		Wait_Calculation, (*Wait For Data Average Calculation V4.A.A.1.6.12*)
		Friction_Remove, (*Wait For Friction Remove V4.A.A.1.6.12*)
		Calibration_Done (*Calibration Done V4.A.A.1.6.12*)
		);
	CAP_CapDisMode_Type :
		( (*V4.A.A.1.7.0*)
		CapDis_Idle,
		CapDis_ProductionInit,
		CapDis_WaitSignal,
		CapDis_WaitCaps,
		CapDis_PrimingReq,
		CapDis_Priming,
		CapDis_Production,
		CapDis_RestartAfterBlock,
		CapDis_RestartAndEmptying,
		CapDis_EmptyingInit,
		CapDis_EmptyingCheck,
		CapDis_Emptying,
		CapDis_EmptyingFault,
		CapDis_EmptyingCycleEnd,
		CapDis_EmptyingDone
		);
	CAP_Type : 	STRUCT
		DataOut : CAP_DataOut_Type;
	END_STRUCT;
	CAP_DataOut_Type : 	STRUCT
		CapperEmpty : BOOL;
		ContainerStop : BOOL; (*//1.63*)
		ReleaseInProduction : BOOL;
		ReleaseInEmptying : BOOL;
		BufferLifted : BOOL;
		ReleaseInManual : BOOL;
		BufferEmpty : BOOL; (*//vrmaCOP*)
		BufferLowered : BOOL;
		BufferHighSpeedReached : BOOL;
		SlowSpeedForEmptyReq : BOOL;
		MachineStop : BOOL;
		MachineStart : BOOL;
		ConfigSaveReq : BOOL;
		GreasingPositioningReq : BOOL;
		UVLampAOn : BOOL; (*v1.4*)
		UVLampBOn : BOOL; (*v1.4*)
		UVLampCOn : BOOL; (*v1.4*)
		Idle : BOOL; (*v1.4*)
		Release1Active : BOOL; (*v1.4*)
		Release2Active : BOOL; (*v1.4*)
		Release3Active : BOOL; (*v1.4*)
		Release4Active : BOOL; (*v1.4*)
		BufferSizeChange_MaxPosition : BOOL; (*//V4.A.A.1.6.11*)
		BufferSizeChange_MinPosition : BOOL; (*//V4.A.A.1.6.11*)
		IonisationBoxDoor : BOOL; (*V4.A.A.1.6.12h*)
		Hopper_TreatmentReq : BOOL; (*v1.7.5*)
		CapDis_MachineRestatBlocked : BOOL; (*V4.A.A.1.7.0*)
		CapDis_MachineAutorestart : BOOL; (*V4.A.A.1.7.0*)
		CapDis_CapsRequest : BOOL; (*V4.A.A.1.7.0*)
		CapDis_EmptyingRequest : BOOL; (*V4.A.A.1.7.0*)
		CapDis_VaporizationRequest : BOOL; (*V4.A.A.1.7.0*)
		CapDis_WarmRequest : BOOL; (*V4.A.A.1.7.0*)
		CapDis_PrimingRequest : BOOL; (*V4.A.A.1.7.0*)
		CapDis_EmptySkip : BOOL; (*V4.A.A.1.7.0*)
		CapDis_InletPreformsStopped : BOOL; (*V4.A.A.1.7.0*)
		CapDis_FillerMode : INT; (*V4.A.A.1.7.0*)
	END_STRUCT;
END_TYPE
```

### COP_Global.typ
```iecst
(*COP*)

TYPE
	COP_Type : 	STRUCT
		DataOut : COP_DataOut_Type;
	END_STRUCT;
	COP_DataOut_Type : 	STRUCT
		RcpActive : BOOL;
		RcpRunning : BOOL;
		RcpDone : BOOL;
		CleaningActive : BOOL;
		CircuitFeeding : BOOL;
		CircuitDrain : BOOL;
		ContainerStop : BOOL;
		RcpManual : BOOL;
		FoamingGunActive : BOOL;
		CapBufferHighSpeedReq : BOOL;
		CapBufferEmptyingReq : BOOL;
		CapChannelEmptyingReq : BOOL;
		CapBufferLiftingReq : BOOL;
		CapBufferLoweringReq : BOOL;
		FixSpeedRequest : BOOL;
		FixSpeedValue : REAL;
		TransferGateCloseReq : BOOL;
		WashingPrdEnable : BOOL;
		WashingPrdNekRinse : BOOL;
		WashingPrdAfterCop : BOOL;
		DisableFillingBottle : BOOL; (*vrmaCOP*)
		CvrEmptyingReq : BOOL;
		DmcInsercionReq : BOOL;
		DmcDisinsercionReq : BOOL;
		MachineStart : BOOL;
		MachineStop : BOOL;
		DmcEnabled : BOOL;
		SmfCleaningValveV : ARRAY[3..10]OF BOOL;
		FlrToProductionHeight : BOOL; (*MASTER NUovo*)
		FlrToMaxMechanicalHeight : BOOL; (*MASTER NUovo*)
		Idle : BOOL;
		ValveWashingCfg : BOOL;
		WashingTray : BOOL;
		SamplingCommand : BOOL;
		SamplingInPosition : BOOL;
		RcpAfterCipEndCfg : BOOL;
		DoserPositioningReq : BOOL; (*v999hema*)
		CopDuringChangeFormatActive : BOOL; (*vrmaCOP*)
		CopValvePurge : BOOL; (*vrmaCOP*)
		CopWipInExecution : BOOL; (*vrmaCOP*)
		CopWashingBeforePurge : BOOL; (*vrmaCOP*)
		CopLapsCounter : BOOL; (*vrmaCOP*)
		CopConAirBlowOffCommand : BOOL; (*vrmaCOP*)
		CopBottleBurstRamp1 : BOOL; (*vrmaCOP*)
		CopPhaseType : USINT;
	END_STRUCT;
END_TYPE
```

### CFG_Global.typ
```iecst
(*CFG*)

TYPE
	CFG_Type : 	STRUCT
		DataOut : CFG_DataOut_Type;
	END_STRUCT;
	CFG_DataOut_Type : 	STRUCT
		Busy : BOOL;
		CapSaved : BOOL;
		OpsSaved : BOOL;
		ConfigLoaded : BOOL;
		OPSDefault : BOOL;
		MotionDefault : BOOL;
		ItcDefault : BOOL;
		PaoDefault : BOOL;
		CfgDefault : BOOL;
		CfgCapDefault : BOOL;
		ErrorSavingMotion : BOOL;
		ErrorSavingItc : BOOL;
		ErrorSavingPao : BOOL;
		ErrorSavingOPS : BOOL;
		ErrorSavingCfg : BOOL;
		ErrorSavingCfgCap : BOOL;
	END_STRUCT;
END_TYPE

(*CONFIGURATION PARAMETER*)

TYPE
	CFG_Par_Type : 	STRUCT
		Filler : CFG_Filler_Type; (*V4.A.A.1.6.12*)
		DummyContainers : CFG_DumCon_Type;
		Cop : CFG_Cop_Type;
		Lifting : CFG_Lifting_Type;
		Process : CFG_Process_Type;
		Machine : CFG_Machine_Type;
		ClosingUnit : CFG_Clu_Type;
		Motors : CFG_Motors_Type;
		WhiteRoom : CFG_WhiteRoom_Type;
		FCI : CFG_FCI_Type;
		ProductChangeOver : CFG_ProductChangeOver_Type;

		Rinser : CFG_RNS_Type;
		CapFedeer : CFG_CFD_Type;
		CapFedeer2 : CFG_CFD_Type; (*v4.A.A.1.7.0*)
		OperatorSafety : CFG_OperatorSafety_Type;
		Maintenance : CFG_MNT_Type;
		Doser : CFG_DOS_Type; (*v999hema*)
	END_STRUCT;
	CFG_Cap_Par_Type : 	STRUCT
		Elements : ARRAY[0..19]OF HMI_ComboBoxElements_Type; (*vrma*)
		Data : ARRAY[0..19]OF CFG_CapFormatData_Type;
	END_STRUCT;
	CFG_Crw_Par_Type : 	STRUCT
		Elements : ARRAY[0..15]OF HMI_ComboBoxElements_Type;
		Data : ARRAY[0..15]OF CFG_CrwFormatData_Type;
	END_STRUCT;
END_TYPE

(*CLOSING UNIT*)

TYPE
	CFG_Clu_Type : 	STRUCT
		Capper : CFG_Cap_Type;
		Crowner : CFG_Crw_Type;
	END_STRUCT;
END_TYPE

(*CAPPER*)

TYPE
	CFG_Cap_Type : 	STRUCT
		GreasingPumpPresent : BOOL;
		Present : BOOL;
		CapDisPresent : BOOL; (*V4.A.A.1.7.0*)
		CapTreatment : BOOL; (*v1.7.5*)
		Buffer : CFG_CapBuffer_Type;
		Channel : CFG_CapChannel_Type;
		Type : CFG_CapManufactor_Type;
		SizeChange : CFG_CapSizeChange_Type;
		HeadRotation : CFG_CapHeadRotation_Type;
		ReleasePresent : USINT; (*1 = Release 1; 2 = Release 2; 3 = Release 3; 4 = Channel 4*)
	END_STRUCT;
	CFG_CapManufactor_Type : 	STRUCT
		Arol : BOOL;
		Zalkin : BOOL;
	END_STRUCT;
	CFG_CapBuffer_Type : 	STRUCT
		Spiral : BOOL;
		Vertical : BOOL;
	END_STRUCT;
	CFG_CapHeadRotation_Type : 	STRUCT
		BrushlessHead : BOOL; (*Arol equatorque or Zalkin Brushless for single head*)
		Hrm : BOOL; (*Brushless for all heads*)
		Drive : BOOL; (*Frequency converter for all heads*)
	END_STRUCT;
	CFG_CapChannel_Type : 	STRUCT
		EmptyThroughPeP : BOOL;
		EmptyThroughGate : BOOL;
		ChannelOptional : ARRAY[0..3]OF CFG_CapChannelOpt_Type;
	END_STRUCT;
	CFG_CapChannelOpt_Type : 	STRUCT
		SlidingSensorPresent : BOOL;
		UvLampLowPressure : BOOL;
		UvLampHonle : BOOL;
		UvLampClaranor : BOOL;
		Ionizer : BOOL;
	END_STRUCT;
	CFG_CamHeighSizeChange_Type : 	STRUCT
		Present : BOOL;
		Manual : BOOL; (*Manual type*)
		Automatic : BOOL; (*Automatic Type*)
	END_STRUCT;
	CFG_CapSizeChange_Type : 	STRUCT  (*Part involved in size change*)
		BottleGuideChange : BOOL; (*Arol Multibody System*)
		BufferSize : BOOL;
		Channel : BOOL;
		CamHeigh : CFG_CamHeighSizeChange_Type;
		PickAndPlace : BOOL;
	END_STRUCT;
	CFG_CapFormatData_Type : 	STRUCT
		HeadRotationDir : BOOL;
		Channel : UINT; (*1 = Channel A; 2 = Channel B; 3 = Channel C; 4 = Channel D*)
		BufferSize : UINT; (*Spiral: 1 = Low Guide Pos; 2 = High Guide Pos;
Vertical: 1 = Width A; 2 = Width B; 3 = Width C; 1 = Width D;*)
		CamHeightPosition : USINT; (* 1 = Low Cam Pos; 2 = High Cam Pos;*)
		PickAndPlaceN : UINT; (*1 = Release 2; 2 = Release 2; 3 = Release 3; 4 = Channel 4*)
	END_STRUCT;
END_TYPE

(*CROWNER*)

TYPE
	CFG_Crw_Type : 	STRUCT
		Present : BOOL;
		Channel : CFG_CrwChannel_Type;
		Type : CFG_CrwManufactor_Type;
	END_STRUCT;
	CFG_CrwChannel_Type : 	STRUCT
		SlidingSensorPresent : BOOL;
		EmptyThroughPeP : BOOL;
		ChannelN : INT;
	END_STRUCT;
	CFG_CrwManufactor_Type : 	STRUCT
		Sidel : BOOL;
		Others : BOOL;
	END_STRUCT;
	CFG_CrwFormatData_Type : 	STRUCT
		Channel : UINT; (*1 = Singol Channel
2 = Double Channel*)
		PickAndPlaceN : UINT;
	END_STRUCT;
END_TYPE

(*DUMMY CONTAINERS*)

TYPE
	CFG_DumCon_Type : 	STRUCT
		DBA_NumValveReadInPosCheck : USINT;
		DBA_NumStepForReversePos : USINT;
		DBA_NumValveInTangSec2 : USINT;
		DBA_NumValveInTangSec1 : USINT;
		Automatic : BOOL;
		Lifting : BOOL;
	END_STRUCT;
END_TYPE

(*COP*)

TYPE
	CFG_Cop_Type : 	STRUCT
		ValveWashing : CFG_ValveWashing_Type;
		FoamingUnitType : CFG_FoamingUnit_Type;
		ChlorinetedWaterBarrierPresent : BOOL;
		DoubleContainerBlock : BOOL;
		CapBufferLifting : BOOL;
		WithSatellites : BOOL;
		DrainableFoamingUnit : BOOL;
		FoamingGunType : CFG_FoamingGun_Type;
		FullFbk : BOOL;
		ExternalDryingOption : BOOL; (*v4.A.A.1.7.0*)
		VenturiRinsing : BOOL;
		ContainerShower : BOOL;
		NeckRinse : BOOL;
	END_STRUCT;
	CFG_ValveWashing_Type : 	STRUCT
		Present : BOOL;
		WithContainers : BOOL;
	END_STRUCT;
	CFG_FoamingGun_Type : 	STRUCT
		WithAVE224 : BOOL;
		WithManualSelector : BOOL;
	END_STRUCT;
	CFG_FoamingUnit_Type : 	STRUCT
		Diversey : BOOL;
		Ecolab : BOOL;
		External : BOOL;
		Loehrke : BOOL;
		Sidel : BOOL;
	END_STRUCT;
END_TYPE

(*LIFTING*)

TYPE
	CFG_Lifting_Type : 	STRUCT
		Present : BOOL; (*V4.A.A.1.6.12*)
		Movements : CFG_LiftingMovement_Type;
		Safety : CFG_LiftingSafety_Type;
	END_STRUCT;
	CFG_LiftingMovement_Type : 	STRUCT
		Filler : CFG_LiftingMovementSku_Type; (*V4.A.A.1.6.12*)
		Crowner : CFG_LiftingMovementClu_Type; (*master nuvo*)
		Capper : CFG_LiftingMovementClu_Type; (*master nuvo*)
		OutletConveyor : CFG_LiftingMovementConveyor_Type; (*V4.A.A.1.6.12*)
		Rinser : CFG_LiftingMovementMotor_Type; (*V4.A.A.1.6.12*)
	END_STRUCT;
	CFG_LiftingMovementConveyor_Type : 	STRUCT
		SizeChangeHeight : BOOL; (*V4.A.A.1.6.12*)
		SizeChangeBottleGuide : BOOL; (*V4.A.A.1.6.12*)
	END_STRUCT;
	CFG_LiftingMovementSku_Type : 	STRUCT
		MaxMechanicalTankHeight : REAL;
		MinMechanicalTankHeight : REAL;
		DeltaTank : REAL;
		MaxMechanicalCammaHeight : REAL;
		MinMechanicalCammaHeight : REAL;
		DeltaCamma : REAL;
		SizeChangeHeight : REAL;
		ToleranceUpCamma : REAL;
		ToleranceDownCamma : REAL;
	END_STRUCT;
	CFG_LiftingMovementClu_Type : 	STRUCT
		SizeChangeHeight : REAL;
		MinMechanicalHeight : REAL;
		MaxMechanicalHeight : REAL;
		Delta : REAL;
		UncouplingRequest : BOOL;
		UncoupledHeight : REAL;
		MaxCoupledHeight : REAL;
	END_STRUCT;
	CFG_LiftingMovementMotor_Type : 	STRUCT
		SizeChangeHeight : REAL;
		MinMechanicalHeight : REAL;
		MaxMechanicalHeight : REAL;
		Delta : REAL;
	END_STRUCT;
	CFG_LiftingSafety_Type : 	STRUCT
		EquipmentSensorHeight : REAL;
	END_STRUCT;
END_TYPE

(*PROCESS*)

TYPE
	CFG_Process_Type : 	STRUCT
		InternalSkid : BOOL;
		BlendFill : BOOL;
	END_STRUCT;
END_TYPE

(*MACHINE*)

TYPE
	CFG_Machine_Type : 	STRUCT
		Type : CFG_MachineModel_Type;
		Combi : CFG_MachineCombi_Type;
	END_STRUCT;
	CFG_MachineModel_Type : 	STRUCT
		SRMA : BOOL;
		SRMB : BOOL;
		SRMC : BOOL;
		SRME : BOOL;
		SRMH : BOOL;
		SRMO : BOOL;
	END_STRUCT;
	CFG_MachineCombi_Type : 	STRUCT
		BAF : BOOL;
		BF : BOOL;
		BLF : BOOL;
		BFL : BOOL;
	END_STRUCT;
END_TYPE

(*MOTORS*)

TYPE
	CFG_Motors_Type : 	STRUCT
		ConveyorVFD : BOOL;
		DoubleInlet : BOOL;
		FootbarPresent : BOOL;
		CoolingFan : CFG_MachineFan_Type;
	END_STRUCT;
	CFG_MachineFan_Type : 	STRUCT
		Inlet : CFG_InletFan_Type;
		Filler : CFG_FillerFan_Type;
		Outlet : CFG_OutletFan_Type;
	END_STRUCT;
	CFG_InletFan_Type : 	STRUCT
		In : ARRAY[1..4]OF CFG_CoolingFan_Type;
		Main : CFG_CoolingFan_Type;
		Out : ARRAY[1..4]OF CFG_CoolingFan_Type;
	END_STRUCT;
	CFG_FillerFan_Type : 	STRUCT
		In : ARRAY[1..10]OF CFG_CoolingFan_Type;
		Main : CFG_CoolingFan_Type;
		Out : ARRAY[1..6]OF CFG_CoolingFan_Type;
	END_STRUCT;
	CFG_OutletFan_Type : 	STRUCT
		In : ARRAY[1..4]OF CFG_CoolingFan_Type;
		Main : CFG_CoolingFan_Type;
		Out : ARRAY[1..4]OF CFG_CoolingFan_Type;
	END_STRUCT;
	CFG_CoolingFan_Type : 	STRUCT
		Present : BOOL;
		CommandPresent : BOOL;
	END_STRUCT;
END_TYPE

(*WHITE ROOM*)

TYPE
	CFG_WhiteRoom_Type : 	STRUCT
		Basement : CFG_WhiteRoomZone_Type;
		Filler : CFG_WhiteRoomZone_Type;
		Rinser : CFG_WhiteRoomZone_Type;
		Transfer : CFG_WhiteRoomZone_Type;
	END_STRUCT;
	CFG_WhiteRoomZone_Type : 	STRUCT
		Present : BOOL;
		NumerOfFan : USINT;
		HmiLightPresent : BOOL;
		GalvaniRoof : BOOL;
	END_STRUCT;
END_TYPE

(*CAPFEEDER - Capfeeder Model*)

TYPE
	CFG_CFD_Type : 	STRUCT
		Aidlin : BOOL;
		Optifeed : BOOL;
		Zalkin : BOOL;
		Customer : BOOL;
	END_STRUCT;
END_TYPE

(*FCI - Full Container Inspector*)

TYPE
	CFG_FCI_Type : 	STRUCT
		FTSystem : BOOL;
		Heuft : BOOL;
		Pressco : BOOL;
		Stratec : BOOL;
		Filltec : BOOL;
		SIS : BOOL;
	END_STRUCT;
END_TYPE

(*PRODUCT CHANGE OVER*)

TYPE
	CFG_ProductChangeOver_Type : 	STRUCT
		APCO : BOOL;
		ICO : BOOL;
	END_STRUCT;
END_TYPE

(*INTERCHANGE SIGNALS*)

TYPE
	CFG_ITC_Type : 	STRUCT
		Blower : ITC_Parameter_Type;
		Labeller : ITC_Parameter_Type;
		Seamer : ITC_Parameter_Type;
		Actis : ITC_Parameter_Type;
		ClosingUnit : ITC_Parameter_Type;
		Skid : ITC_Parameter_Type;
		CoreBlend : ITC_Parameter_Type;
		Cip : ITC_Parameter_Type;
		Cop : ITC_Parameter_Type;
		WhiteRoom : ITC_Parameter_Type;
		InletConveyors : ITC_Parameter_Type;
		OutletConveyors : ITC_Parameter_Type;
		Fci : ITC_Parameter_Type;
		Vbc : ITC_Parameter_Type;
		CapFeeder1 : ITC_Parameter_Type;
		CapFeeder2 : ITC_Parameter_Type;
		Coder : ITC_Parameter_Type;
		LidFeeder : ITC_Parameter_Type;
		SignalConcentrator : ITC_Parameter_Type;
		DataAcquisition : ITC_Parameter_Type;
		ProductChangeover : ITC_Parameter_Type;
		SikoMultibody : ITC_Parameter_Type; (*V4.A.A.1.6.12*)
		RinserRecSkd : ITC_Parameter_Type; (*V4.A.A.1.6.12*)
		FlavorDoser : ITC_Parameter_Type; (*V4.A.A.1.6.12*)
		CapDis : ITC_Parameter_Type; (*V4.A.A.1.7.0*)
		DoserHema : ITC_Parameter_Type; (*v999hema*)
	END_STRUCT;
	ITC_Parameter_Type : 	STRUCT
		ComType : USINT; (*Communication Type:
0 = NOT PRESENT
1 = TCP IP
2 = ETH IP
3 = MODBUS TCP
4 = PROFIBUS
5 = POWERLINK EPL
6 = HW
7 = UDP
8 = SCC
9 = PROFINET
10 = OPC*)
		ComAddress : STRING[35]; (*Communication Partner Adress*)
		ComSwap : BOOL; (*Swap the comunication*)
		EnableServer : BOOL; (*Select Mode: SERVER = TRUE / CLIENT = FALSE*)
		LocalPort : UINT; (*Local port number used to Receive*)
		RemotePort : UINT; (*Remote port number used o Send*)
		RecLength : UDINT; (*Received data Length (BYTE)*)
		SendLength : UDINT; (*Send data Length (BYTE)*)
		RecTimeOut : TIME; (*Receive data TimeOut [ms]*)
		SendTimeAct : TIME; (*Send data Time [ms]*)
	END_STRUCT;
END_TYPE

(*FILLER V4.A.A.1.6.12*)

TYPE
	CFG_Filler_Type : 	STRUCT
		ContainerLifting : BOOL;
	END_STRUCT;
END_TYPE

(*RINSER*)

TYPE
	CFG_RNS_Type : 	STRUCT
		Present : BOOL;
		PressureNozzleControlInsertion : BOOL; (*vrma*)
		PressureNozzleControlContinous : BOOL; (*vrma*)
		Recovery : BOOL;
		NoBottleNoSpray : BOOL; (*Master nuovo*)
		ExternalRecoverySkid : BOOL; (*V4.A.A.1.6.12*)
		CipPresent : BOOL; (*V4.A.A.1.7.0*)
		FootbarPresent : BOOL; (*V4.A.A.1.7.0*)
	END_STRUCT;
END_TYPE

(*OPERATOR SAETY*)

TYPE
	CFG_OPS_Type : 	STRUCT
		Door : ARRAY[0..MAX_CFG_DoorConfiguration]OF CFG_Doors_Type;
		Jog : ARRAY[0..MAX_CFG_JogConfiguration]OF CFG_Jog_Type;
		Emergency : ARRAY[0..MAX_CFG_EmergencyConfiguration]OF CFG_Emergency_Type;
		Layout : CFG_Layout_Type; (*V 1.61*)
	END_STRUCT;
	CFG_Doors_Type : 	STRUCT
		Number : UINT;
		Zone : UINT;
	END_STRUCT;
	CFG_Jog_Type : 	STRUCT
		Zone : UINT;
	END_STRUCT;
	CFG_Emergency_Type : 	STRUCT
		Number : UINT;
	END_STRUCT;
	CFG_Layout_Type : 	STRUCT  (*V 1.61*)
		StarsNumber : UINT;
		SidesNumber : UINT;
		ExitLenght : UINT;
		BufferDoorPosition : UINT; (*V4.A.A.1.6.12d*)
	END_STRUCT;
END_TYPE

(*CONFIGURATION*)

TYPE
	CFG_OperatorSafety_Type : 	STRUCT
		AcknoledgeButtonZone : BOOL;
		DoorCabinet : BOOL; (*v1.4 DoorCabinet Sensor Presence*)
		EuchnerKey : BOOL; (*v1.4 Euchner key Presence*)
	END_STRUCT;
END_TYPE

(*MAINTENANCE*)

TYPE
	CFG_MNT_Type : 	STRUCT
		DeEnergization : BOOL; (*LOTO*)
		PreventiveMaintenance : BOOL; (*TPM*)
	END_STRUCT;
END_TYPE

(*DOSER v999hema*)

TYPE
	CFG_DOS_Type : 	STRUCT
		Present : BOOL;
		RecoverySkid : BOOL;
	END_STRUCT;
END_TYPE
```

### CRW_Global.typ
```iecst
TYPE
	CRW_Config_Type : 	STRUCT
		Channel1 : BOOL;
		Channel2 : BOOL;
		PickAndPlace : UINT;
		Hopper1 : REAL;
		Hopper2 : REAL;
	END_STRUCT;
	CRW_Mode_Type :
		(
		CRW_Idle,
		CRW_Production,
		CRW_ProductionReady,
		CRW_Emptying
		);
END_TYPE

(*CROWNER*)

TYPE
	CRW_Type : 	STRUCT
		DataOut : CRW_DataOut_Type;
	END_STRUCT;
	CRW_DataOut_Type : 	STRUCT
		ReleaseInProduction : BOOL;
		ReleaseInEmptying : BOOL;
		ReleaseInManual : BOOL;
		SlowSpeedForEmptyReq : BOOL;
		ConfigSaveReq : BOOL;
		HeadRinsingReq : BOOL;
		ContainerStop : BOOL;
		Idle : BOOL;
		MachineStart : BOOL; (*vrmaCOP*)
		ChannelEmptyingReq : BOOL; (*vrmaCOP*)
		ChannelEmpty : BOOL; (*vrmaCOP*)
	END_STRUCT;
END_TYPE
```

### CSR_Global.typ
```iecst
(*CSR*)

TYPE
	CSR_Type : 	STRUCT
		DataOut : CSR_DataOut_Type;
	END_STRUCT;
	CSR_DataOut_Type : 	STRUCT
		AutoSizeChangeActive : BOOL; (*MASTER NUovo*)
		Active : BOOL;
		CipPosition : BOOL;
		ProductionPosition : BOOL;
		LiftingEnableSafetyRequ : BOOL;
		SkfStop : BOOL;
		SkfStart : BOOL;
		Idle : BOOL; (*v1.4*)
		ContainerStop : BOOL; (*//1.63*)
		PositioningInProgress : BOOL; (*V4.A.A.1.6.12*)
		PositioningDone : BOOL; (*V4.A.A.1.6.12*)
		CrwPositioningReq : BOOL; (*V4.A.A.1.7.0*)
		CapPositioningReq : BOOL; (*V4.A.A.1.7.0*)
		MachineStop : BOOL; (*V4.A.A.1.7.0*)
		SkfTargetPosition : REAL;
		StartCopAfterChangeOver : BOOL; (*v999 cop test*)
		CopDuringChangeFormatReq : BOOL; (*v999 cop test*)
		CapperPositionUncoupled : BOOL; (*MASTER NUovo*)
		FlrToMaxMechanicalHeightDone : BOOL; (*MASTER NUovo*)
		FlrCipPositionHeightDone : BOOL;
		FlrAndCamHeightControlOk : BOOL; (*v999*)
		FlrPrdPositionHeightDone : BOOL; (*MASTER NUovo*)
	END_STRUCT;
END_TYPE

(*SKF_SCU*)

TYPE
	SKF_SCU_Type : 	STRUCT
		DataOut : SKF_SCU_DataOut_Type;
	END_STRUCT;
	SKF_SCU_DataOut_Type : 	STRUCT
		Actuator_1_Position : REAL; (*Actuator 1 position [mm]*)
		Actuator_2_Position : REAL; (*Actuator 2 position [mm]*)
		Actuator_3_Position : REAL; (*Actuator 3 position [mm]*)
		Actuator_Position_Offset : REAL; (*Offset --> Difference from Real Position and Actuator Position [mm]*)
		Running : BOOL;
		InitializationDone : BOOL;
		Idle : BOOL; (*v1.4*)
	END_STRUCT;
	CSR_Lift_SeqMode_Type :
		(
		CSR_LiftIdle,
		CSR_LiftBottlesStop,
		CSR_LiftMachineStop,
		CSR_LiftRaiseMaximumHeight,
		CSR_LiftNewSize,
		CSR_LiftDescentSizeHeight,
		CSR_LiftWaitSelectorOff,
		CSR_LiftManualMode
		);
	CSR_Sequencer_Type :
		(
		CSR_Idle := 0,
		CSR_WaitSafetyEnable := 205,
		CSR_SizeChangeHeightRequ := 210,
		CSR_SizeChangeHeightDone := 220,
		CSR_SizeChangeProdHeightRequ := 222,
		CSR_SizeChangeProdHeightDone := 240,
		CSR_SizeChangeCipHeightRequ := 260,
		CSR_SizeChangeCipHeightDone := 262,
		CSR_ManualWaitSafetyEnable := 605,
		CSR_ManualMode := 606,
		CSR_ManualModeTank := 610,
		CSR_ManualModeCamma := 620,
		CSR_MaxMechanicalHeightRequ := 621,
		CSR_MaxMechanicalHeightDone := 622,
		CSR_Fault := 9999
		);
END_TYPE
```

### DMC_Global.typ
```iecst
TYPE
	DMC_Mode_Type : 	STRUCT
		AutomaticMode : DMC_Status_Type;
		ManualMode : DMC_Status_Type;
	END_STRUCT;
	DMC_Status_Type : 	STRUCT
		CycleActive : BOOL;
		CycleAborted : BOOL;
		SecondHalfPositionDone : BOOL;
		SecondHalfRotToProdDone : BOOL;
		SecondHalfRotToCipDone : BOOL;
		FirstHalfRotToProdDone : BOOL;
		FirstHalfRotToCipDone : BOOL;
		SecondHalfPistonUpDone : BOOL;
		SecondHalfPistonDownDone : BOOL;
		FirstHalfPistonUpDone : BOOL;
		FirstHalfPistonDownDone : BOOL;
		SecondHalfCheckToProdDone : BOOL;
		FirstHalfCheckToProdDone : BOOL;
		SecondHalfCheckToCipDone : BOOL;
		FirstHalfCheckToCipDone : BOOL;
		FirstHalfPositionDone : BOOL;
		FirstHalfDmcRemoved : BOOL;
		FirstHalfDmcInserted : BOOL;
		SecondHalfDmcRemoved : BOOL;
		SecondHalfDmcInserted : BOOL;
	END_STRUCT;
	DMC_ModeManualSequencerType :
		(
		DMC_ManWait := 0,
		DMC_ManFillerFirstHalfPosReq := 1, (*v999*)
		DMC_ManDummyFirstHalfWaitPosDone := 2,
		DMC_ManDiscargeAirForDownMov := 3, (*v999*)
		DMC_ManFirstSecCommandSelection := 4,
		DMC_ManFirstSectorRotToCip := 5,
		DMC_ManFirstSectorRotToProd := 6,
		DMC_ManCommandDummyBottleUp := 7,
		DMC_ManDummyContWaitComCheckSec1 := 8,
		DMC_ManDummyContDinsControl := 9,
		DMC_ManDmcFirstHalfInsErrFilStop := 10,
		DMC_ManReturnToFirstHalfPosition := 11,
		DMC_ManReturnToFirstWaitPosDone := 12,
		DMC_ManFirstHalfCheck := 13,
		DMC_ManFirstHalfCheckConfToRest := 14,
		DMC_ManFirstHalfDisWaitPressOk := 15,
		DMC_ManDmcFirstHalfInstFillStop := 16,
		DMC_ManFillerSecondHalfPosReq := 17,
		DMC_ManDmcSecondHalfWaitPosDone := 18,
		DMC_ManDiscargeAirForDownMovSec2 := 19,
		DMC_ManSecondSecCommandSelection := 20,
		DMC_ManSecondSectorRotToCip := 21,
		DMC_ManSecondSectorRotToProd := 22,
		DMC_ManCommandDummyBottleUpSec2 := 23,
		DMC_ManDummyContWaitComCheckSec2 := 24,
		DMC_ManDummyContDinsControlSec2 := 25,
		DMC_ManDmcHalfInsErrFilStopSec2 := 26,
		DMC_ManReturnToSecondHalfPos := 27,
		DMC_ManReturnToSecondWaitPosDone := 28,
		DMC_ManSecondHalfCheck := 29,
		DMC_ManSecondHalfCheckConfToRest := 30,
		DMC_ManSecondHalfDisWaitPressOk := 31,
		DMC_ManDmcSecondHalfInstFillStop := 32,
		DMC_MauFaultPistonDownSec1 := 33,
		DMC_MauFaultPistonDownSec2 := 34,
		DMC_ManFaultRotToCipSec1 := 35,
		DMC_ManFaultRotToCipSec2 := 36,
		DMC_ManFaultRotToProdSec1 := 37,
		DMC_ManFaultRotToProdSec2 := 38,
		DMC_ManFault := 99
		);
	DMC_SequencerType :
		(
		DMC_Wait := 0,
		DMC_WaitMachineEmptyAndSlowDown := 1,
		DMC_LftCenteringCupUp := 2,
		DMC_DummyContInstalling := 4,
		DMC_DummyContInstalledControl := 5,
		DMC_DummyContInsMachineStop := 6,
		DMC_DummyContInsCsrPositioning := 7,
		DMC_DummyContInsLftCenterCupDown := 8,
		DMC_DummyContInsFmcCipMode := 9,
		DMC_DummyContInstalled := 10,
		DMC_DummyContDisMachineStop := 11,
		DMC_DummyContDisFmcCenterCupUp := 12,
		DMC_DummyContDisLftCenterCupUp := 13,
		DMC_DummyContDisCsrPositioning := 14,
		DMC_DummyContDisMachineStart := 15,
		DMC_DummyContDisinsection := 16,
		DMC_DummyContDinsControl := 17,
		DMC_DummyContRemovedDone := 18,
		DMC_TankAndCammaHeigthControl := 19, (*v999*)
		DMC_FillerHeightPositionReq := 20, (*v999*)
		DMC_FillerFirstHalfPosReq := 21, (*v999*)
		DMC_CommandDummyBottleDown := 22, (*v999*)
		DMC_WaitMachineStopped := 23, (*v999*)
		DMC_DiscargeAirForDownMovement := 24, (*v999*)
		DMC_CommandDummyBottleUp := 25, (*v999*)
		DMC_FillerSecondHalfPosReq := 26, (*v999*)
		DMC_DiscargeSecHalfAirForDownMov := 27, (*v999*)
		DMC_SecondHalfComDummyBottleDown := 28, (*v999*)
		DMC_SecondHalfDummyContInstCont := 29, (*v999*)
		DMC_FillerFirstHalfPosReqForDis := 30, (*v999*)
		DMC_DiscargeAirForDownMovForDis := 31, (*v999*)
		DMC_CommandDummyBottleDownForDis := 32, (*v999*)
		DMC_CommandDummyBottleUpForDis := 33, (*v999*)
		DMC_FillerSecondHalfPosReqForDis := 34, (*v999*)
		DMC_SecHalfComDumBotDownForDis := 35, (*v999*)
		DMC_CommandDummyBotUpSecondHalf := 36, (*v999*)
		DMC_SecondHalfDmcInstCont := 37, (*v999*)
		DMC_FillerSecondHalfPosReqforDis := 38, (*v999*)
		DMC_DiscargeAirSecHalfForDownMov := 39,
		DMC_SecHalfComDummyBottleDownDis := 40,
		DMC_CommandDummyBottleUpDis := 41,
		DMC_SecondHalfDummyContDisCont := 42,
		DMC_DMCFirstHalfInstMachineStop := 43,
		DMC_FisrtHalfWaitFillerStop := 44,
		DMC_ReturnToFirstHalfPosition := 46,
		DMC_DMCFirstHalfInsErrFilStop := 45,
		DMC_FirstHalfCheck := 47,
		DMC_DMCSecondHalfInstMachineStop := 48,
		DMC_DummyContSecondHalfInstCont := 49,
		DMC_DMCSecondHalfInsErrFilStop := 50,
		DMC_ReturnToSecondHalfPosition := 51,
		DMC_SecondHalfCheck := 52,
		DMC_FirstHalfDisReverseForCheck := 53,
		DMC_FirstHalDisWaitCheckDone := 54,
		DMC_SecondHalfDisReverseForCheck := 55,
		DMC_SecondHalDisWaitCheckDone := 56,
		DMC_DummyGenericErrorDownToCip := 57,
		DMC_FirstHalfDisWaitPressureOk := 58,
		DMC_SecondHalfDisWaitPressureOk := 59,
		DMC_FirstHalfInsWaitPressureOk := 60,
		DMC_FirstHalfCheckConfToRestart := 61,
		DMC_SecondHalfCheckConfToRestart := 62,
		DMC_DMCFirstHalfDisMachineStop := 64,
		DMC_SecondHalfInsWaitPressureOk := 63,
		DMC_FirstHalfDisCheckToRestart := 65,
		DMC_SecondHalfDisCheck := 66,
		DMC_SecondHalfDisCheckToRestart := 67,
		DMC_DummyErrorDownToCipSec2 := 68,
		DMC_DummyErrorDownToProdSec1 := 69,
		DMC_DummyErrorDownToProdSec2 := 70,
		DMC_DummyFirstHalfWaitPosDone := 71,
		DMC_DummySecondHalfWaitPosDone := 72,
		DMC_DummySecHalfDisWaitPosDone := 73,
		DMC_FillerSecHalfDisWaitFillStop := 75,
		DMC_DummyFirstHalfDisWaitPosDone := 74,
		DMC_ReturnToFirstWaitPosDone := 76,
		DMC_ReturnToSecondHalfPosDone := 77,
		DMC_FirstHalfDisRevPosDone := 78,
		DMC_SecondHalfDisRevPosDone := 79,
		DMC_CycleAbortedChooseStep := 81,
		DMC_CycleAbortedCheckContidion := 80,
		DMC_WaitConditionForAborting := 82,
		DMC_ReturnToProdHeight := 83,
		DMC_Fault := 99
		);
END_TYPE
```
